C01813=1094.520,430.598,-102.360,178.831,24.503,153.665
C01814=1094.514,430.353,-102.317,178.828,24.492,153.663
C01815=1094.508,430.106,-102.276,178.825,24.481,153.660
C01816=1094.502,429.860,-102.233,178.822,24.469,153.658
C01817=1094.495,429.613,-102.192,178.819,24.459,153.656
C01818=1094.490,429.367,-102.149,178.817,24.448,153.653
C01819=1094.483,429.120,-102.107,178.813,24.437,153.651
C01820=1094.477,428.875,-102.065,178.811,24.426,153.649
C01821=1094.470,428.628,-102.023,178.808,24.416,153.646
C01822=1094.464,428.382,-101.981,178.805,24.405,153.644
C01823=1094.457,428.135,-101.939,178.802,24.394,153.642
C01824=1094.451,427.889,-101.898,178.799,24.383,153.639
C01825=1094.445,427.643,-101.855,178.797,24.373,153.637
C01826=1094.439,427.397,-101.814,178.793,24.362,153.635
C01827=1094.433,427.150,-101.772,178.791,24.352,153.633
C01828=1094.426,426.904,-101.730,178.788,24.342,153.630
C01829=1094.420,426.658,-101.688,178.785,24.331,153.628
C01830=1094.413,426.411,-101.646,178.782,24.320,153.626
C01831=1094.407,426.165,-101.605,178.779,24.310,153.624
C01832=1094.401,425.919,-101.563,178.776,24.300,153.622
C01833=1094.395,425.672,-101.522,178.774,24.289,153.619
C01834=1094.389,425.443,-101.483,178.771,24.280,153.617
C01835=1094.384,425.215,-101.444,178.768,24.270,153.615
C01836=1094.378,424.987,-101.406,178.766,24.261,153.613
C01837=1094.372,424.758,-101.367,178.763,24.251,153.611
C01838=1094.366,424.529,-101.329,178.760,24.242,153.609
C01839=1094.360,424.301,-101.290,178.757,24.232,153.607
C01840=1094.355,424.073,-101.252,178.755,24.223,153.605
C01841=1094.349,423.844,-101.213,178.752,24.214,153.603
C01842=1094.344,423.598,-101.172,178.749,24.204,153.601
C01843=1094.337,423.351,-101.130,178.746,24.194,153.599
C01844=1094.330,423.105,-101.089,178.744,24.184,153.597
C01845=1094.324,422.859,-101.047,178.741,24.174,153.595
C01846=1094.319,422.612,-101.007,178.738,24.164,153.593
C01847=1094.312,422.365,-100.965,178.734,24.154,153.591
C01848=1094.306,422.119,-100.923,178.732,24.144,153.589
C01849=1094.300,421.873,-100.883,178.729,24.134,153.587
C01850=1094.294,421.627,-100.842,178.726,24.125,153.585
C01851=1094.287,421.380,-100.800,178.723,24.115,153.583
C01852=1094.281,421.134,-100.759,178.720,24.105,153.581
C01853=1094.275,420.887,-100.718,178.717,24.095,153.579
C01854=1094.269,420.641,-100.677,178.714,24.086,153.577
C01855=1094.263,420.393,-100.636,178.712,24.076,153.575
C01856=1094.256,420.147,-100.595,178.709,24.067,153.573
C01857=1094.250,419.901,-100.553,178.706,24.057,153.571
C01858=1094.245,419.654,-100.513,178.703,24.048,153.569
C01859=1094.238,419.408,-100.472,178.700,24.038,153.567
C01860=1094.232,419.161,-100.431,178.697,24.029,153.565
C01861=1094.225,418.914,-100.391,178.694,24.019,153.563
C01862=1094.219,418.668,-100.349,178.691,24.010,153.561
C01863=1094.214,418.421,-100.308,178.689,24.000,153.559
C01864=1094.207,418.175,-100.268,178.686,23.991,153.557
C01865=1094.201,417.929,-100.227,178.683,23.982,153.555
C01866=1094.195,417.682,-100.187,178.680,23.972,153.553
C01867=1094.189,417.436,-100.145,178.677,23.963,153.551
C01868=1094.183,417.188,-100.104,178.675,23.954,153.549
C01869=1094.176,416.942,-100.064,178.672,23.945,153.548
C01870=1094.171,416.695,-100.023,178.669,23.936,153.546
C01871=1094.164,416.449,-99.982,178.666,23.926,153.544
C01872=1094.158,416.202,-99.942,178.663,23.918,153.542
C01873=1094.152,415.956,-99.901,178.660,23.908,153.540
C01874=1094.146,415.709,-99.861,178.657,23.899,153.538
C01875=1094.140,415.462,-99.821,178.654,23.890,153.536
C01876=1094.134,415.216,-99.780,178.652,23.882,153.535
C01877=1094.128,414.969,-99.740,178.649,23.873,153.533
C01878=1094.122,414.723,-99.700,178.646,23.864,153.531
C01879=1094.114,414.476,-99.658,178.643,23.855,153.529
C01880=1094.109,414.229,-99.618,178.640,23.846,153.527
C01881=1094.102,413.983,-99.577,178.636,23.837,153.526
C01882=1094.096,413.735,-99.538,178.634,23.828,153.524
C01883=1094.091,413.489,-99.497,178.631,23.820,153.522
C01884=1094.084,413.242,-99.457,178.628,23.811,153.520
C01885=1094.078,412.996,-99.417,178.625,23.802,153.519
C01886=1094.071,412.749,-99.377,178.623,23.794,153.517
C01887=1094.066,412.502,-99.336,178.620,23.785,153.515
C01888=1094.059,412.256,-99.296,178.617,23.776,153.513
C01889=1094.053,412.009,-99.256,178.614,23.768,153.512
C01890=1094.048,411.788,-99.221,178.611,23.760,153.510
C01891=1094.043,411.567,-99.184,178.609,23.753,153.509
C01892=1094.038,411.345,-99.148,178.606,23.745,153.507
C01893=1094.032,411.125,-99.112,178.604,23.737,153.506
C01894=1094.026,410.904,-99.076,178.601,23.730,153.504
C01895=1094.021,410.682,-99.041,178.599,23.722,153.503
C01896=1094.015,410.461,-99.004,178.595,23.714,153.501
C01897=1094.011,410.240,-98.969,178.593,23.706,153.499
C01898=1094.004,409.993,-98.929,178.591,23.698,153.498
C01899=1093.998,409.746,-98.889,178.588,23.690,153.496
C01900=1093.992,409.500,-98.849,178.584,23.681,153.495
C01901=1093.986,409.253,-98.808,178.582,23.673,153.493
C01902=1093.980,409.006,-98.769,178.579,23.665,153.491
C01903=1093.974,408.759,-98.729,178.576,23.656,153.490
C01904=1093.968,408.513,-98.690,178.574,23.648,153.488
C01905=1093.962,408.266,-98.650,178.570,23.640,153.486
C01906=1093.956,408.019,-98.610,178.568,23.632,153.485
C01907=1093.949,407.773,-98.570,178.565,23.624,153.483
C01908=1093.943,407.525,-98.531,178.561,23.616,153.482
C01909=1093.938,407.279,-98.491,178.559,23.607,153.480
C01910=1093.932,407.032,-98.451,178.556,23.599,153.478
C01911=1093.926,406.785,-98.411,178.554,23.591,153.477
C01912=1093.920,406.538,-98.372,178.550,23.583,153.475
C01913=1093.914,406.291,-98.332,178.547,23.575,153.474
C01914=1093.908,406.045,-98.293,178.545,23.567,153.472
C01915=1093.902,405.798,-98.253,178.542,23.559,153.470
C01916=1093.895,405.551,-98.214,178.539,23.551,153.469
C01917=1093.889,405.304,-98.174,178.536,23.543,153.467
C01918=1093.883,405.058,-98.135,178.533,23.536,153.466
C01919=1093.877,404.811,-98.096,178.530,23.528,153.464
C01920=1093.871,404.564,-98.056,178.528,23.520,153.463
C01921=1093.865,404.317,-98.017,178.524,23.512,153.461
C01922=1093.859,404.071,-97.977,178.522,23.504,153.460
C01923=1093.853,403.824,-97.938,178.519,23.497,153.458
C01924=1093.847,403.577,-97.899,178.516,23.489,153.457
C01925=1093.841,403.330,-97.860,178.513,23.481,153.455
C01926=1093.835,403.083,-97.820,178.510,23.474,153.454
C01927=1093.829,402.836,-97.781,178.507,23.466,153.452
C01928=1093.823,402.590,-97.742,178.505,23.458,153.451
C01929=1093.817,402.343,-97.703,178.501,23.450,153.449
C01930=1093.811,402.096,-97.664,178.499,23.443,153.448
C01931=1093.805,401.849,-97.625,178.496,23.435,153.446
C01932=1093.799,401.602,-97.585,178.493,23.428,153.445
C01933=1093.792,401.355,-97.546,178.490,23.421,153.444
C01934=1093.787,401.108,-97.508,178.487,23.412,153.442
C01935=1093.781,400.861,-97.468,178.485,23.405,153.441
C01936=1093.775,400.614,-97.429,178.482,23.398,153.439
C01937=1093.769,400.368,-97.391,178.479,23.390,153.438
C01938=1093.763,400.121,-97.351,178.476,23.383,153.437
C01939=1093.757,399.874,-97.312,178.473,23.376,153.435
C01940=1093.751,399.627,-97.274,178.470,23.368,153.434
C01941=1093.745,399.380,-97.235,178.468,23.361,153.432
C01942=1093.739,399.133,-97.195,178.464,23.353,153.431
C01943=1093.733,398.886,-97.157,178.462,23.346,153.430
C01944=1093.727,398.639,-97.118,178.459,23.339,153.428
C01945=1093.720,398.393,-97.079,178.456,23.332,153.427
C01946=1093.715,398.172,-97.044,178.453,23.325,153.426
C01947=1093.710,397.951,-97.010,178.451,23.319,153.424
C01948=1093.704,397.730,-96.976,178.448,23.312,153.423
C01949=1093.700,397.509,-96.941,178.446,23.306,153.422
C01950=1093.694,397.289,-96.907,178.443,23.299,153.421
C01951=1093.688,397.068,-96.872,178.441,23.293,153.420
C01952=1093.683,396.847,-96.837,178.438,23.287,153.418
C01953=1093.678,396.626,-96.803,178.435,23.280,153.417
C01954=1093.671,396.379,-96.764,178.433,23.274,153.416
C01955=1093.666,396.132,-96.726,178.430,23.266,153.415
C01956=1093.659,395.885,-96.687,178.427,23.259,153.413
C01957=1093.654,395.638,-96.649,178.424,23.252,153.412
C01958=1093.647,395.391,-96.610,178.421,23.245,153.411
C01959=1093.642,395.144,-96.572,178.418,23.238,153.409
C01960=1093.636,394.898,-96.533,178.415,23.231,153.408
C01961=1093.630,394.650,-96.494,178.413,23.224,153.407
C01962=1093.624,394.404,-96.457,178.410,23.217,153.406
C01963=1093.618,394.157,-96.418,178.406,23.210,153.404
C01964=1093.612,393.910,-96.379,178.404,23.203,153.403
C01965=1093.606,393.663,-96.342,178.401,23.197,153.402
C01966=1093.600,393.416,-96.303,178.398,23.190,153.401
C01967=1093.594,393.169,-96.265,178.395,23.183,153.399
C01968=1093.588,392.922,-96.226,178.392,23.176,153.398
C01969=1093.582,392.675,-96.189,178.389,23.169,153.397
C01970=1093.576,392.428,-96.151,178.387,23.163,153.396
C01971=1093.570,392.181,-96.111,178.384,23.156,153.394
C01972=1093.564,391.934,-96.074,178.380,23.149,153.393
C01973=1093.558,391.688,-96.036,178.378,23.142,153.392
C01974=1093.552,391.440,-95.998,178.375,23.136,153.391
C01975=1093.546,391.193,-95.960,178.372,23.130,153.390
C01976=1093.540,390.947,-95.922,178.369,23.123,153.388
C01977=1093.534,390.699,-95.884,178.366,23.116,153.387
C01978=1093.528,390.452,-95.846,178.363,23.110,153.386
C01979=1093.522,390.206,-95.807,178.360,23.103,153.385
C01980=1093.516,389.959,-95.769,178.357,23.096,153.384
C01981=1093.510,389.712,-95.732,178.355,23.090,153.383
C01982=1093.504,389.465,-95.694,178.351,23.083,153.381
C01983=1093.498,389.218,-95.656,178.348,23.076,153.380
C01984=1093.491,388.971,-95.618,178.345,23.070,153.379
C01985=1093.486,388.724,-95.581,178.343,23.064,153.378
C01986=1093.480,388.477,-95.543,178.340,23.057,153.377
C01987=1093.474,388.230,-95.505,178.337,23.051,153.376
C01988=1093.468,387.983,-95.468,178.333,23.044,153.375
C01989=1093.462,387.736,-95.429,178.331,23.038,153.373
C01990=1093.456,387.489,-95.392,178.328,23.031,153.372
C01991=1093.450,387.242,-95.354,178.325,23.025,153.371
C01992=1093.444,386.995,-95.317,178.322,23.019,153.370
C01993=1093.438,386.748,-95.279,178.319,23.013,153.369
C01994=1093.432,386.502,-95.241,178.316,23.006,153.368
C01995=1093.426,386.254,-95.203,178.314,23.000,153.367
C01996=1093.420,386.007,-95.166,178.310,22.993,153.366
C01997=1093.414,385.760,-95.128,178.307,22.987,153.365
C01998=1093.408,385.513,-95.091,178.304,22.981,153.363
C01999=1093.402,385.267,-95.053,178.301,22.975,153.362
C02000=1093.397,385.019,-95.016,178.298,22.969,153.361
C02001=1093.391,384.772,-94.978,178.296,22.962,153.360
C02002=1093.386,384.558,-94.946,178.294,22.957,153.359
C02003=1093.381,384.343,-94.913,178.290,22.951,153.358
C02004=1093.376,384.129,-94.880,178.288,22.946,153.357
C02005=1093.371,383.915,-94.848,178.285,22.940,153.356
C02006=1093.365,383.700,-94.816,178.283,22.935,153.356
C02007=1093.361,383.486,-94.783,178.281,22.930,153.355
C02008=1093.355,383.272,-94.751,178.278,22.924,153.354
C02009=1093.351,383.057,-94.719,178.276,22.919,153.353
C02010=1093.345,382.811,-94.681,178.273,22.913,153.352
C02011=1093.339,382.563,-94.644,178.270,22.907,153.351
C02012=1093.332,382.316,-94.607,178.267,22.901,153.350
C02013=1093.326,382.069,-94.569,178.264,22.895,153.349
C02014=1093.321,381.821,-94.532,178.261,22.889,153.348
C02015=1093.314,381.575,-94.495,178.258,22.883,153.347
C02016=1093.308,381.328,-94.458,178.255,22.877,153.346
C02017=1093.303,381.080,-94.421,178.252,22.871,153.345
C02018=1093.296,380.834,-94.384,178.249,22.866,153.344
C02019=1093.291,380.587,-94.347,178.245,22.859,153.343
C02020=1093.285,380.339,-94.310,178.242,22.853,153.342
C02021=1093.278,380.093,-94.273,178.239,22.847,153.341
C02022=1093.273,379.845,-94.236,178.237,22.841,153.340
C02023=1093.267,379.598,-94.199,178.234,22.836,153.339
C02024=1093.261,379.351,-94.162,178.231,22.830,153.338
C02025=1093.255,379.104,-94.125,178.228,22.824,153.337
C02026=1093.249,378.857,-94.087,178.226,22.818,153.336
C02027=1093.243,378.610,-94.051,178.222,22.813,153.335
C02028=1093.237,378.362,-94.014,178.219,22.807,153.334
C02029=1093.231,378.115,-93.977,178.217,22.801,153.333
C02030=1093.225,377.868,-93.940,178.213,22.796,153.332
C02031=1093.220,377.621,-93.903,178.210,22.790,153.331
C02032=1093.213,377.374,-93.867,178.208,22.784,153.330
C02033=1093.208,377.127,-93.830,178.204,22.778,153.329
C02034=1093.202,376.880,-93.794,178.202,22.772,153.328
C02035=1093.197,376.633,-93.757,178.198,22.767,153.327
C02036=1093.191,376.385,-93.720,178.196,22.761,153.326
C02037=1093.185,376.138,-93.683,178.192,22.755,153.325
C02038=1093.179,375.891,-93.646,178.189,22.749,153.324
C02039=1093.173,375.644,-93.610,178.186,22.744,153.323
C02040=1093.167,375.396,-93.573,178.183,22.738,153.323
C02041=1093.161,375.150,-93.537,178.180,22.732,153.322
C02042=1093.156,374.903,-93.500,178.177,22.727,153.321
C02043=1093.149,374.656,-93.463,178.175,22.722,153.320
C02044=1093.144,374.408,-93.426,178.172,22.716,153.319
C02045=1093.138,374.160,-93.390,178.169,22.710,153.318
C02046=1093.132,373.913,-93.353,178.166,22.705,153.317
C02047=1093.126,373.666,-93.317,178.163,22.699,153.316
C02048=1093.120,373.420,-93.281,178.160,22.694,153.315
C02049=1093.115,373.172,-93.244,178.157,22.688,153.315
C02050=1093.108,372.925,-93.208,178.154,22.683,153.314
C02051=1093.102,372.678,-93.172,178.150,22.677,153.313
C02052=1093.096,372.431,-93.135,178.147,22.672,153.312
C02053=1093.091,372.183,-93.099,178.145,22.667,153.311
C02054=1093.084,371.936,-93.062,178.142,22.661,153.310
C02055=1093.078,371.689,-93.026,178.139,22.656,153.309
C02056=1093.073,371.441,-92.990,178.136,22.650,153.309
C02057=1093.067,371.194,-92.953,178.133,22.645,153.308
C02058=1093.057,370.793,-92.895,178.128,22.636,153.306
C02059=1093.048,370.391,-92.836,178.123,22.627,153.305
C02060=1093.038,369.990,-92.777,178.119,22.619,153.304
C02061=1093.029,369.590,-92.719,178.114,22.610,153.302
C02062=1093.023,369.342,-92.683,178.111,22.605,153.301
C02063=1093.017,369.094,-92.647,178.107,22.600,153.301
C02064=1093.011,368.847,-92.610,178.104,22.594,153.300
C02065=1093.005,368.600,-92.575,178.101,22.589,153.299
C02066=1092.999,368.353,-92.538,178.099,22.584,153.298
C02067=1092.993,368.105,-92.503,178.096,22.579,153.297
C02068=1092.988,367.858,-92.467,178.092,22.574,153.297
C02069=1092.982,367.611,-92.430,178.089,22.568,153.296
C02070=1092.976,367.363,-92.394,178.086,22.563,153.295
C02071=1092.971,367.116,-92.359,178.084,22.558,153.294
C02072=1092.964,366.869,-92.323,178.081,22.553,153.293
C02073=1092.958,366.622,-92.287,178.077,22.548,153.293
C02074=1092.954,366.374,-92.251,178.074,22.542,153.292
C02075=1092.948,366.127,-92.215,178.071,22.537,153.291
C02076=1092.941,365.880,-92.179,178.069,22.532,153.290
C02077=1092.936,365.633,-92.143,178.066,22.527,153.289
C02078=1092.930,365.385,-92.108,178.062,22.522,153.289
C02079=1092.924,365.137,-92.072,178.059,22.517,153.288
C02080=1092.918,364.890,-92.037,178.056,22.512,153.287
C02081=1092.912,364.643,-92.000,178.054,22.507,153.287
C02082=1092.906,364.396,-91.964,178.050,22.502,153.286
C02083=1092.900,364.149,-91.929,178.047,22.497,153.285
C02084=1092.894,363.901,-91.893,178.044,22.491,153.284
C02085=1092.889,363.654,-91.858,178.042,22.487,153.284
C02086=1092.883,363.406,-91.822,178.038,22.482,153.283
C02087=1092.876,363.159,-91.787,178.035,22.477,153.282
C02088=1092.871,362.912,-91.752,178.032,22.471,153.281
C02089=1092.865,362.664,-91.716,178.029,22.467,153.281
C02090=1092.859,362.417,-91.681,178.026,22.462,153.280
C02091=1092.853,362.170,-91.645,178.023,22.457,153.279
C02092=1092.847,361.922,-91.609,178.020,22.452,153.279
C02093=1092.842,361.675,-91.574,178.017,22.447,153.278
C02094=1092.836,361.427,-91.538,178.014,22.442,153.277
C02095=1092.831,361.180,-91.503,178.011,22.437,153.276
C02096=1092.824,360.932,-91.468,178.008,22.433,153.276
C02097=1092.818,360.685,-91.433,178.005,22.428,153.275
C02098=1092.812,360.438,-91.397,178.002,22.423,153.274
C02099=1092.807,360.191,-91.362,177.999,22.418,153.274
C02100=1092.801,359.943,-91.326,177.996,22.414,153.273
C02101=1092.795,359.695,-91.292,177.993,22.408,153.272
C02102=1092.789,359.448,-91.256,177.990,22.403,153.271
C02103=1092.783,359.200,-91.221,177.987,22.399,153.271
C02104=1092.778,358.953,-91.185,177.984,22.394,153.270
C02105=1092.771,358.705,-91.151,177.980,22.389,153.270
C02106=1092.766,358.458,-91.115,177.978,22.385,153.269
C02107=1092.760,358.211,-91.080,177.975,22.380,153.268
C02108=1092.754,357.963,-91.046,177.971,22.375,153.267
C02109=1092.748,357.716,-91.010,177.969,22.371,153.267
C02110=1092.739,357.330,-90.955,177.963,22.363,153.266
C02111=1092.730,356.944,-90.901,177.959,22.356,153.265
C02112=1092.721,356.558,-90.846,177.955,22.349,153.264
C02113=1092.712,356.172,-90.791,177.950,22.342,153.263
C02114=1092.706,355.925,-90.757,177.947,22.337,153.262
C02115=1092.700,355.678,-90.722,177.943,22.332,153.261
C02116=1092.695,355.429,-90.687,177.941,22.328,153.261
C02117=1092.688,355.183,-90.652,177.937,22.323,153.260
C02118=1092.683,354.935,-90.617,177.934,22.318,153.260
C02119=1092.677,354.688,-90.582,177.932,22.314,153.259
C02120=1092.671,354.440,-90.547,177.928,22.309,153.258
C02121=1092.666,354.192,-90.512,177.925,22.304,153.258
C02122=1092.659,353.945,-90.478,177.922,22.300,153.257
C02123=1092.654,353.697,-90.443,177.919,22.295,153.256
C02124=1092.648,353.449,-90.408,177.916,22.291,153.256
C02125=1092.642,353.203,-90.373,177.913,22.286,153.255
C02126=1092.637,352.955,-90.339,177.910,22.282,153.255
C02127=1092.631,352.707,-90.304,177.907,22.277,153.254
C02128=1092.625,352.460,-90.269,177.904,22.273,153.253
C02129=1092.619,352.212,-90.234,177.901,22.269,153.253
C02130=1092.613,351.965,-90.200,177.898,22.264,153.252
C02131=1092.608,351.717,-90.166,177.894,22.259,153.252
C02132=1092.601,351.470,-90.130,177.892,22.255,153.251
C02133=1092.595,351.222,-90.096,177.889,22.250,153.250
C02134=1092.586,350.816,-90.040,177.884,22.243,153.249
C02135=1092.576,350.409,-89.983,177.879,22.236,153.249
C02136=1092.566,350.002,-89.926,177.874,22.229,153.248
C02137=1092.557,349.596,-89.870,177.869,22.221,153.247
C02138=1092.552,349.348,-89.835,177.865,22.217,153.246
C02139=1092.546,349.101,-89.801,177.863,22.213,153.245
C02140=1092.540,348.853,-89.767,177.859,22.208,153.245
C02141=1092.534,348.605,-89.732,177.856,22.204,153.244
C02142=1092.529,348.358,-89.698,177.853,22.199,153.244
C02143=1092.523,348.111,-89.664,177.851,22.195,153.243
C02144=1092.518,347.863,-89.629,177.847,22.191,153.243
C02145=1092.511,347.615,-89.595,177.844,22.187,153.242
C02146=1092.505,347.368,-89.561,177.841,22.182,153.242
C02147=1092.500,347.120,-89.526,177.838,22.178,153.241
C02148=1092.494,346.873,-89.492,177.835,22.174,153.241
C02149=1092.488,346.625,-89.458,177.832,22.169,153.240
C02150=1092.482,346.377,-89.424,177.829,22.165,153.239
C02151=1092.477,346.129,-89.390,177.825,22.161,153.239
C02152=1092.471,345.882,-89.356,177.823,22.157,153.238
C02153=1092.465,345.635,-89.322,177.819,22.152,153.238
C02154=1092.459,345.387,-89.287,177.817,22.148,153.237
C02155=1092.453,345.139,-89.254,177.813,22.144,153.237
C02156=1092.448,344.891,-89.219,177.811,22.140,153.236
C02157=1092.442,344.644,-89.185,177.807,22.135,153.236
C02158=1092.436,344.408,-89.153,177.805,22.132,153.235
C02159=1092.431,344.172,-89.120,177.802,22.128,153.235
C02160=1092.426,343.935,-89.088,177.798,22.124,153.234
C02161=1092.420,343.700,-89.056,177.796,22.119,153.234
C02162=1092.414,343.464,-89.023,177.793,22.116,153.233
C02163=1092.408,343.229,-88.991,177.790,22.112,153.233
C02164=1092.403,342.992,-88.959,177.787,22.108,153.232
C02165=1092.398,342.756,-88.927,177.784,22.104,153.232
C02166=1092.392,342.509,-88.893,177.781,22.100,153.231
C02167=1092.386,342.260,-88.859,177.778,22.096,153.231
C02168=1092.380,342.013,-88.825,177.775,22.092,153.230
C02169=1092.375,341.765,-88.792,177.772,22.088,153.230
C02170=1092.369,341.518,-88.758,177.769,22.084,153.229
C02171=1092.363,341.270,-88.724,177.766,22.079,153.229
C02172=1092.357,341.023,-88.690,177.763,22.075,153.228
C02173=1092.352,340.775,-88.657,177.759,22.071,153.228
C02174=1092.346,340.527,-88.623,177.757,22.067,153.227
C02175=1092.340,340.280,-88.589,177.753,22.063,153.227
C02176=1092.334,340.032,-88.555,177.751,22.059,153.226
C02177=1092.328,339.784,-88.522,177.747,22.055,153.226
C02178=1092.322,339.536,-88.488,177.744,22.051,153.225
C02179=1092.317,339.288,-88.454,177.742,22.047,153.225
C02180=1092.311,339.041,-88.421,177.738,22.043,153.225
C02181=1092.305,338.793,-88.387,177.735,22.039,153.224
C02182=1092.300,338.545,-88.354,177.732,22.035,153.224
C02183=1092.294,338.298,-88.321,177.729,22.031,153.223
C02184=1092.288,338.051,-88.287,177.726,22.027,153.223
C02185=1092.282,337.803,-88.253,177.723,22.023,153.222
C02186=1092.277,337.555,-88.220,177.720,22.019,153.222
C02187=1092.271,337.307,-88.187,177.717,22.015,153.221
C02188=1092.265,337.060,-88.153,177.714,22.011,153.221
C02189=1092.259,336.812,-88.120,177.710,22.007,153.220
C02190=1092.253,336.564,-88.087,177.708,22.003,153.220
C02191=1092.248,336.316,-88.053,177.704,21.999,153.220
C02192=1092.242,336.068,-88.020,177.701,21.995,153.219
C02193=1092.236,335.821,-87.986,177.698,21.992,153.219
C02194=1092.230,335.573,-87.953,177.695,21.988,153.218
C02195=1092.225,335.325,-87.920,177.692,21.984,153.218
C02196=1092.219,335.078,-87.886,177.689,21.980,153.217
C02197=1092.213,334.830,-87.854,177.686,21.976,153.217
C02198=1092.207,334.582,-87.820,177.683,21.972,153.216
C02199=1092.202,334.334,-87.787,177.680,21.969,153.216
C02200=1092.195,334.087,-87.754,177.677,21.965,153.216
C02201=1092.190,333.839,-87.721,177.674,21.961,153.215
C02202=1092.184,333.591,-87.688,177.671,21.957,153.215
C02203=1092.179,333.343,-87.654,177.668,21.954,153.214
C02204=1092.172,333.095,-87.622,177.664,21.949,153.214
C02205=1092.167,332.848,-87.589,177.661,21.946,153.214
C02206=1092.162,332.600,-87.555,177.659,21.942,153.213
C02207=1092.156,332.353,-87.522,177.655,21.938,153.213
C02208=1092.150,332.105,-87.489,177.652,21.934,153.212
C02209=1092.144,331.857,-87.456,177.650,21.930,153.212
C02210=1092.138,331.609,-87.423,177.646,21.927,153.212
C02211=1092.132,331.362,-87.390,177.643,21.923,153.211
C02212=1092.126,331.114,-87.357,177.640,21.920,153.211
C02213=1092.120,330.866,-87.324,177.637,21.915,153.210
C02214=1092.111,330.477,-87.273,177.632,21.910,153.210
C02215=1092.102,330.087,-87.222,177.628,21.905,153.209
C02216=1092.093,329.698,-87.170,177.623,21.898,153.209
C02217=1092.083,329.308,-87.119,177.618,21.893,153.208
C02218=1092.078,329.061,-87.085,177.615,21.889,153.208
C02219=1092.072,328.813,-87.053,177.611,21.885,153.207
C02220=1092.066,328.565,-87.021,177.608,21.882,153.207
C02221=1092.061,328.318,-86.988,177.605,21.879,153.207
C02222=1092.054,328.070,-86.955,177.602,21.874,153.206
C02223=1092.049,327.821,-86.922,177.599,21.871,153.206
C02224=1092.043,327.574,-86.889,177.596,21.868,153.205
C02225=1092.036,327.326,-86.857,177.593,21.864,153.205
C02226=1092.031,327.078,-86.824,177.590,21.860,153.205
C02227=1092.026,326.831,-86.792,177.587,21.857,153.204
C02228=1092.020,326.583,-86.760,177.584,21.853,153.204
C02229=1092.014,326.335,-86.726,177.580,21.849,153.204
C02230=1092.008,326.086,-86.694,177.577,21.846,153.203
C02231=1092.002,325.839,-86.662,177.575,21.842,153.203
C02232=1091.996,325.592,-86.629,177.571,21.838,153.203
C02233=1091.991,325.343,-86.597,177.568,21.835,153.202
C02234=1091.984,325.096,-86.564,177.565,21.832,153.202
C02235=1091.978,324.848,-86.532,177.563,21.828,153.201
C02236=1091.974,324.600,-86.500,177.559,21.824,153.201
C02237=1091.968,324.352,-86.467,177.556,21.821,153.201
C02238=1091.962,324.104,-86.435,177.553,21.817,153.200
C02239=1091.956,323.857,-86.402,177.550,21.814,153.200
C02240=1091.951,323.609,-86.370,177.547,21.810,153.200
C02241=1091.945,323.360,-86.338,177.544,21.807,153.199
C02242=1091.938,323.113,-86.305,177.541,21.803,153.199
C02243=1091.933,322.865,-86.273,177.538,21.800,153.199
C02244=1091.927,322.617,-86.240,177.534,21.796,153.198
C02245=1091.921,322.369,-86.208,177.532,21.792,153.198
C02246=1091.916,322.122,-86.176,177.529,21.789,153.198
C02247=1091.910,321.873,-86.144,177.526,21.786,153.197
C02248=1091.904,321.626,-86.111,177.522,21.782,153.197
C02249=1091.899,321.378,-86.079,177.519,21.779,153.197
C02250=1091.893,321.130,-86.047,177.517,21.775,153.196
C02251=1091.888,320.882,-86.016,177.514,21.772,153.196
C02252=1091.881,320.635,-85.983,177.510,21.768,153.196
C02253=1091.876,320.386,-85.950,177.507,21.764,153.195
C02254=1091.871,320.139,-85.919,177.504,21.761,153.195
C02255=1091.865,319.890,-85.887,177.502,21.758,153.195
C02256=1091.859,319.643,-85.855,177.498,21.754,153.194
C02257=1091.853,319.395,-85.823,177.495,21.751,153.194
C02258=1091.848,319.148,-85.790,177.492,21.747,153.194
C02259=1091.842,318.900,-85.758,177.489,21.744,153.193
C02260=1091.837,318.651,-85.726,177.486,21.741,153.193
C02261=1091.831,318.404,-85.694,177.483,21.737,153.193
C02262=1091.825,318.155,-85.662,177.480,21.733,153.192
C02263=1091.820,317.908,-85.630,177.477,21.730,153.192
C02264=1091.814,317.660,-85.598,177.474,21.727,153.192
C02265=1091.808,317.412,-85.567,177.470,21.723,153.191
C02266=1091.799,317.016,-85.515,177.466,21.718,153.191
C02267=1091.791,316.620,-85.465,177.461,21.712,153.190
C02268=1091.782,316.224,-85.413,177.456,21.706,153.190
C02269=1091.773,315.827,-85.363,177.452,21.702,153.189
C02270=1091.767,315.579,-85.331,177.448,21.698,153.189
C02271=1091.761,315.332,-85.300,177.445,21.694,153.189
C02272=1091.755,315.083,-85.268,177.442,21.691,153.189
C02273=1091.750,314.836,-85.236,177.439,21.688,153.188
C02274=1091.744,314.587,-85.205,177.436,21.685,153.188
C02275=1091.739,314.339,-85.173,177.433,21.682,153.188
C02276=1091.732,314.092,-85.142,177.430,21.678,153.187
C02277=1091.727,313.844,-85.110,177.427,21.675,153.187
C02278=1091.721,313.596,-85.078,177.424,21.672,153.187
C02279=1091.715,313.347,-85.047,177.421,21.668,153.187
C02280=1091.709,313.100,-85.016,177.418,21.665,153.186
C02281=1091.703,312.852,-84.984,177.415,21.662,153.186
C02282=1091.698,312.604,-84.952,177.411,21.659,153.186
C02283=1091.691,312.356,-84.921,177.408,21.655,153.186
C02284=1091.686,312.108,-84.890,177.405,21.652,153.185
C02285=1091.680,311.861,-84.858,177.402,21.649,153.185
C02286=1091.674,311.612,-84.827,177.399,21.646,153.185
C02287=1091.669,311.364,-84.795,177.396,21.643,153.185
C02288=1091.663,311.116,-84.763,177.393,21.639,153.184
C02289=1091.657,310.868,-84.733,177.390,21.636,153.184
C02290=1091.651,310.620,-84.701,177.387,21.633,153.184
C02291=1091.645,310.373,-84.669,177.384,21.630,153.183
C02292=1091.640,310.125,-84.639,177.381,21.627,153.183
C02293=1091.634,309.877,-84.607,177.378,21.623,153.183
C02294=1091.628,309.629,-84.577,177.375,21.621,153.183
C02295=1091.622,309.381,-84.545,177.371,21.617,153.183
C02296=1091.617,309.133,-84.514,177.368,21.614,153.182
C02297=1091.611,308.885,-84.483,177.365,21.611,153.182
C02298=1091.605,308.636,-84.451,177.362,21.608,153.182
C02299=1091.599,308.389,-84.420,177.359,21.604,153.182
C02300=1091.594,308.141,-84.389,177.356,21.602,153.181
C02301=1091.588,307.893,-84.357,177.353,21.598,153.181
C02302=1091.582,307.645,-84.327,177.350,21.595,153.181
C02303=1091.577,307.398,-84.295,177.347,21.591,153.181
C02304=1091.570,307.149,-84.265,177.344,21.589,153.180
C02305=1091.565,306.902,-84.233,177.341,21.585,153.180
C02306=1091.559,306.654,-84.203,177.338,21.582,153.180
C02307=1091.553,306.405,-84.171,177.335,21.579,153.180
C02308=1091.547,306.158,-84.140,177.332,21.576,153.179
C02309=1091.542,305.910,-84.109,177.329,21.573,153.179
C02310=1091.537,305.661,-84.078,177.326,21.570,153.179
C02311=1091.530,305.414,-84.047,177.322,21.567,153.179
C02312=1091.525,305.165,-84.016,177.319,21.563,153.178
C02313=1091.519,304.918,-83.986,177.316,21.560,153.178
C02314=1091.514,304.669,-83.955,177.313,21.557,153.178
C02315=1091.508,304.422,-83.923,177.310,21.554,153.178
C02316=1091.502,304.173,-83.892,177.307,21.551,153.177
C02317=1091.497,303.926,-83.862,177.304,21.548,153.177
C02318=1091.488,303.532,-83.813,177.299,21.543,153.177
C02319=1091.479,303.138,-83.763,177.295,21.538,153.176
C02320=1091.470,302.746,-83.715,177.289,21.533,153.176
C02321=1091.461,302.352,-83.667,177.285,21.528,153.176
C02322=1091.455,302.103,-83.636,177.282,21.525,153.175
C02323=1091.449,301.856,-83.604,177.279,21.522,153.175
C02324=1091.444,301.608,-83.574,177.275,21.519,153.175
C02325=1091.439,301.360,-83.543,177.272,21.515,153.175
C02326=1091.433,301.112,-83.513,177.269,21.513,153.175
C02327=1091.427,300.864,-83.482,177.266,21.509,153.174
C02328=1091.422,300.616,-83.451,177.263,21.506,153.174
C02329=1091.416,300.368,-83.421,177.260,21.503,153.174
C02330=1091.410,300.119,-83.390,177.257,21.500,153.174
C02331=1091.405,299.871,-83.359,177.254,21.497,153.173
C02332=1091.399,299.624,-83.329,177.251,21.494,153.173
C02333=1091.394,299.376,-83.298,177.248,21.491,153.173
C02334=1091.388,299.128,-83.268,177.245,21.488,153.173
C02335=1091.383,298.880,-83.237,177.242,21.485,153.173
C02336=1091.377,298.631,-83.207,177.239,21.482,153.172
C02337=1091.371,298.383,-83.177,177.236,21.479,153.172
C02338=1091.366,298.135,-83.146,177.233,21.476,153.172
C02339=1091.361,297.887,-83.115,177.231,21.473,153.172
C02340=1091.355,297.640,-83.085,177.227,21.469,153.171
C02341=1091.349,297.392,-83.055,177.224,21.467,153.171
C02342=1091.342,297.143,-83.024,177.221,21.464,153.171
C02343=1091.337,296.895,-82.994,177.218,21.461,153.171
C02344=1091.332,296.647,-82.963,177.214,21.458,153.171
C02345=1091.326,296.399,-82.933,177.211,21.455,153.171
C02346=1091.320,296.151,-82.903,177.209,21.452,153.170
C02347=1091.315,295.903,-82.873,177.206,21.449,153.170
C02348=1091.309,295.655,-82.843,177.202,21.446,153.170
C02349=1091.303,295.407,-82.812,177.199,21.443,153.170
C02350=1091.297,295.159,-82.782,177.196,21.440,153.170
C02351=1091.292,294.911,-82.752,177.193,21.437,153.169
C02352=1091.286,294.663,-82.722,177.190,21.434,153.169
C02353=1091.280,294.415,-82.692,177.187,21.431,153.169
C02354=1091.275,294.167,-82.662,177.184,21.429,153.169
C02355=1091.269,293.919,-82.632,177.181,21.426,153.169
C02356=1091.263,293.670,-82.602,177.178,21.423,153.169
C02357=1091.257,293.422,-82.572,177.175,21.420,153.168
C02358=1091.252,293.174,-82.541,177.172,21.417,153.168
C02359=1091.247,292.926,-82.511,177.169,21.414,153.168
C02360=1091.241,292.678,-82.481,177.166,21.411,153.168
C02361=1091.236,292.430,-82.451,177.163,21.408,153.168
C02362=1091.230,292.182,-82.421,177.160,21.406,153.167
C02363=1091.224,291.934,-82.392,177.157,21.403,153.167
C02364=1091.218,291.686,-82.361,177.154,21.400,153.167
C02365=1091.212,291.437,-82.332,177.151,21.397,153.167
C02366=1091.206,291.190,-82.301,177.148,21.394,153.167
C02367=1091.201,290.941,-82.272,177.145,21.391,153.167
C02368=1091.195,290.693,-82.241,177.142,21.388,153.166
C02369=1091.190,290.445,-82.212,177.139,21.385,153.166
C02370=1091.181,290.065,-82.166,177.134,21.381,153.166
C02371=1091.172,289.686,-82.121,177.129,21.377,153.166
C02372=1091.164,289.306,-82.075,177.125,21.372,153.165
C02373=1091.155,288.927,-82.029,177.120,21.368,153.165
C02374=1091.149,288.679,-82.000,177.117,21.365,153.165
C02375=1091.144,288.430,-81.970,177.114,21.362,153.165
C02376=1091.137,288.182,-81.941,177.111,21.359,153.165
C02377=1091.132,287.934,-81.911,177.108,21.356,153.165
C02378=1091.126,287.686,-81.881,177.105,21.354,153.165
C02379=1091.121,287.437,-81.851,177.102,21.351,153.164
C02380=1091.114,287.189,-81.822,177.099,21.348,153.164
C02381=1091.108,286.942,-81.792,177.096,21.345,153.164
C02382=1091.103,286.693,-81.762,177.093,21.342,153.164
C02383=1091.098,286.445,-81.733,177.090,21.340,153.164
C02384=1091.092,286.197,-81.704,177.087,21.337,153.163
C02385=1091.086,285.949,-81.674,177.083,21.334,153.163
C02386=1091.080,285.701,-81.644,177.080,21.331,153.163
C02387=1091.075,285.453,-81.614,177.077,21.328,153.163
C02388=1091.069,285.204,-81.585,177.074,21.326,153.163
C02389=1091.063,284.956,-81.556,177.071,21.323,153.163
C02390=1091.058,284.708,-81.526,177.069,21.320,153.163
C02391=1091.052,284.460,-81.497,177.066,21.318,153.163
C02392=1091.047,284.212,-81.468,177.063,21.315,153.162
C02393=1091.041,283.963,-81.438,177.060,21.312,153.162
C02394=1091.035,283.715,-81.409,177.057,21.309,153.162
C02395=1091.030,283.467,-81.380,177.054,21.306,153.162
C02396=1091.024,283.219,-81.350,177.051,21.303,153.162
C02397=1091.018,282.971,-81.321,177.048,21.301,153.162
C02398=1091.013,282.722,-81.291,177.044,21.298,153.161
C02399=1091.007,282.474,-81.262,177.041,21.295,153.161
C02400=1091.001,282.226,-81.233,177.038,21.292,153.161
C02401=1090.996,281.978,-81.204,177.035,21.289,153.161
C02402=1090.990,281.730,-81.174,177.032,21.287,153.161
C02403=1090.984,281.481,-81.145,177.029,21.284,153.161
C02404=1090.979,281.234,-81.116,177.027,21.282,153.161
C02405=1090.973,280.986,-81.087,177.024,21.279,153.160
C02406=1090.968,280.736,-81.058,177.021,21.276,153.160
C02407=1090.962,280.488,-81.029,177.018,21.273,153.160
C02408=1090.957,280.241,-80.999,177.015,21.271,153.160
C02409=1090.950,279.992,-80.970,177.011,21.268,153.160
C02410=1090.945,279.744,-80.941,177.008,21.265,153.160
C02411=1090.939,279.495,-80.912,177.005,21.262,153.160
C02412=1090.934,279.248,-80.883,177.002,21.259,153.159
C02413=1090.928,278.999,-80.854,176.999,21.257,153.159
C02414=1090.922,278.751,-80.824,176.997,21.255,153.159
C02415=1090.917,278.503,-80.796,176.994,21.252,153.159
C02416=1090.911,278.255,-80.767,176.991,21.249,153.159
C02417=1090.905,278.006,-80.738,176.988,21.246,153.159
C02418=1090.899,277.758,-80.709,176.985,21.244,153.159
C02419=1090.894,277.510,-80.680,176.981,21.241,153.159
C02420=1090.888,277.262,-80.651,176.978,21.238,153.159
C02421=1090.883,277.013,-80.621,176.975,21.235,153.158
C02422=1090.874,276.643,-80.579,176.970,21.231,153.158
C02423=1090.866,276.273,-80.536,176.967,21.228,153.158
C02424=1090.857,275.903,-80.493,176.962,21.224,153.158
C02425=1090.848,275.533,-80.450,176.957,21.220,153.158
C02426=1090.843,275.285,-80.421,176.954,21.217,153.158
C02427=1090.838,275.036,-80.393,176.951,21.214,153.157
C02428=1090.831,274.788,-80.364,176.949,21.212,153.157
C02429=1090.827,274.540,-80.335,176.946,21.209,153.157
C02430=1090.820,274.292,-80.306,176.943,21.206,153.157
C02431=1090.815,274.044,-80.278,176.940,21.204,153.157
C02432=1090.809,273.795,-80.249,176.937,21.201,153.157
C02433=1090.804,273.546,-80.220,176.933,21.199,153.157
C02434=1090.798,273.298,-80.192,176.930,21.196,153.157
C02435=1090.792,273.050,-80.163,176.928,21.194,153.157
C02436=1090.787,272.802,-80.135,176.925,21.191,153.156
C02437=1090.781,272.554,-80.106,176.922,21.188,153.156
C02438=1090.775,272.305,-80.077,176.919,21.185,153.156
C02439=1090.770,272.057,-80.049,176.916,21.183,153.156
C02440=1090.764,271.809,-80.020,176.912,21.180,153.156
C02441=1090.758,271.561,-79.992,176.909,21.177,153.156
C02442=1090.752,271.312,-79.964,176.907,21.175,153.156
C02443=1090.747,271.064,-79.934,176.904,21.172,153.156
C02444=1090.741,270.816,-79.906,176.901,21.170,153.156
C02445=1090.736,270.567,-79.878,176.898,21.167,153.155
C02446=1090.730,270.319,-79.849,176.894,21.165,153.155
C02447=1090.724,270.071,-79.821,176.891,21.162,153.155
C02448=1090.719,269.823,-79.793,176.889,21.160,153.155
C02449=1090.713,269.574,-79.765,176.886,21.157,153.155
C02450=1090.708,269.325,-79.736,176.883,21.154,153.155
C02451=1090.702,269.077,-79.707,176.880,21.152,153.155
C02452=1090.696,268.829,-79.679,176.876,21.149,153.155
C02453=1090.691,268.580,-79.651,176.873,21.146,153.155
C02454=1090.685,268.332,-79.623,176.871,21.144,153.155
C02455=1090.679,268.084,-79.595,176.868,21.141,153.154
C02456=1090.673,267.835,-79.566,176.865,21.139,153.154
C02457=1090.668,267.587,-79.538,176.862,21.136,153.154
C02458=1090.662,267.339,-79.509,176.859,21.134,153.154
C02459=1090.656,267.091,-79.481,176.856,21.131,153.154
C02460=1090.651,266.843,-79.453,176.853,21.129,153.154
C02461=1090.645,266.594,-79.425,176.850,21.126,153.154
C02462=1090.640,266.346,-79.397,176.847,21.123,153.154
C02463=1090.634,266.097,-79.369,176.844,21.121,153.154
C02464=1090.628,265.849,-79.341,176.841,21.118,153.154
C02465=1090.623,265.600,-79.312,176.838,21.116,153.153
C02466=1090.617,265.352,-79.284,176.835,21.113,153.153
C02467=1090.611,265.103,-79.256,176.832,21.111,153.153
C02468=1090.606,264.855,-79.228,176.829,21.108,153.153
C02469=1090.601,264.607,-79.200,176.826,21.105,153.153
C02470=1090.595,264.359,-79.172,176.824,21.103,153.153
C02471=1090.589,264.111,-79.145,176.820,21.101,153.153
C02472=1090.583,263.862,-79.116,176.817,21.098,153.153
C02473=1090.577,263.614,-79.088,176.814,21.095,153.153
C02474=1090.569,263.246,-79.047,176.810,21.092,153.153
C02475=1090.560,262.879,-79.006,176.805,21.088,153.153
C02476=1090.551,262.512,-78.966,176.801,21.084,153.152
C02477=1090.543,262.145,-78.924,176.797,21.081,153.152
C02478=1090.537,261.896,-78.896,176.794,21.078,153.152
C02479=1090.531,261.648,-78.868,176.790,21.076,153.152
C02480=1090.526,261.399,-78.841,176.787,21.073,153.152
C02481=1090.520,261.151,-78.813,176.785,21.071,153.152
C02482=1090.514,260.903,-78.785,176.782,21.069,153.152
C02483=1090.508,260.654,-78.757,176.779,21.066,153.152
C02484=1090.502,260.405,-78.730,176.776,21.063,153.152
C02485=1090.497,260.157,-78.702,176.773,21.061,153.152
C02486=1090.491,259.909,-78.674,176.770,21.059,153.152
C02487=1090.485,259.660,-78.647,176.767,21.056,153.152
C02488=1090.479,259.412,-78.619,176.764,21.054,153.152
C02489=1090.474,259.163,-78.591,176.761,21.052,153.152
C02490=1090.468,258.915,-78.564,176.758,21.049,153.152
C02491=1090.462,258.666,-78.536,176.755,21.046,153.151
C02492=1090.457,258.418,-78.508,176.752,21.044,153.151
C02493=1090.451,258.170,-78.481,176.749,21.041,153.151
C02494=1090.445,257.921,-78.453,176.746,21.039,153.151
C02495=1090.440,257.673,-78.426,176.743,21.037,153.151
C02496=1090.434,257.425,-78.398,176.740,21.034,153.151
C02497=1090.429,257.175,-78.371,176.737,21.032,153.151
C02498=1090.422,256.928,-78.343,176.735,21.029,153.151
C02499=1090.417,256.679,-78.316,176.731,21.027,153.151
C02500=1090.411,256.431,-78.289,176.728,21.024,153.151
C02501=1090.406,256.182,-78.261,176.725,21.021,153.151
C02502=1090.400,255.934,-78.233,176.723,21.019,153.151
C02503=1090.395,255.685,-78.206,176.720,21.017,153.151
C02504=1090.389,255.437,-78.178,176.716,21.014,153.150
C02505=1090.383,255.188,-78.151,176.713,21.012,153.150
C02506=1090.378,254.940,-78.123,176.711,21.010,153.150
C02507=1090.372,254.692,-78.097,176.708,21.007,153.150
C02508=1090.367,254.443,-78.070,176.705,21.004,153.150
C02509=1090.360,254.195,-78.042,176.702,21.002,153.150
C02510=1090.355,253.946,-78.015,176.699,21.000,153.150
C02511=1090.350,253.698,-77.987,176.696,20.997,153.150
C02512=1090.344,253.450,-77.960,176.693,20.995,153.150
C02513=1090.338,253.200,-77.932,176.690,20.993,153.150
C02514=1090.333,252.952,-77.906,176.687,20.990,153.150
C02515=1090.327,252.704,-77.878,176.684,20.987,153.150
C02516=1090.321,252.456,-77.851,176.681,20.985,153.150
C02517=1090.316,252.207,-77.824,176.679,20.983,153.150
C02518=1090.310,251.959,-77.796,176.676,20.980,153.150
C02519=1090.305,251.710,-77.769,176.672,20.978,153.150
C02520=1090.299,251.461,-77.742,176.670,20.975,153.149
C02521=1090.294,251.213,-77.715,176.667,20.973,153.149
C02522=1090.288,250.964,-77.688,176.664,20.970,153.149
C02523=1090.283,250.716,-77.660,176.661,20.967,153.149
C02524=1090.277,250.468,-77.634,176.658,20.965,153.149
C02525=1090.271,250.220,-77.607,176.655,20.963,153.149
C02526=1090.263,249.849,-77.566,176.650,20.959,153.149
C02527=1090.255,249.479,-77.526,176.647,20.956,153.149
C02528=1090.247,249.108,-77.486,176.642,20.952,153.149
C02529=1090.238,248.739,-77.446,176.638,20.948,153.149
C02530=1090.233,248.490,-77.419,176.635,20.945,153.148
C02531=1090.227,248.242,-77.392,176.633,20.944,153.148
C02532=1090.222,247.993,-77.365,176.629,20.941,153.148
C02533=1090.217,247.745,-77.338,176.626,20.938,153.148
C02534=1090.211,247.496,-77.311,176.623,20.936,153.148
C02535=1090.205,247.247,-77.284,176.621,20.934,153.148
C02536=1090.199,246.998,-77.257,176.618,20.931,153.148
C02537=1090.194,246.750,-77.231,176.615,20.928,153.148
C02538=1090.189,246.501,-77.203,176.612,20.926,153.148
C02539=1090.183,246.253,-77.177,176.609,20.924,153.148
C02540=1090.177,246.005,-77.150,176.606,20.922,153.148
C02541=1090.171,245.756,-77.124,176.604,20.919,153.148
C02542=1090.166,245.508,-77.096,176.600,20.917,153.148
C02543=1090.160,245.259,-77.070,176.597,20.914,153.148
C02544=1090.155,245.011,-77.043,176.595,20.912,153.148
C02545=1090.149,244.763,-77.016,176.592,20.909,153.148
C02546=1090.144,244.513,-76.990,176.589,20.907,153.147
C02547=1090.138,244.265,-76.963,176.586,20.905,153.147
C02548=1090.133,244.017,-76.937,176.583,20.903,153.147
C02549=1090.127,243.768,-76.910,176.580,20.900,153.147
C02550=1090.121,243.520,-76.883,176.578,20.898,153.147
C02551=1090.115,243.271,-76.857,176.574,20.895,153.147
C02552=1090.111,243.022,-76.830,176.571,20.893,153.147
C02553=1090.105,242.774,-76.803,176.569,20.891,153.147
C02554=1090.099,242.525,-76.777,176.566,20.888,153.147
C02555=1090.093,242.277,-76.750,176.563,20.886,153.147
C02556=1090.088,242.028,-76.724,176.560,20.884,153.147
C02557=1090.082,241.780,-76.698,176.557,20.881,153.147
C02558=1090.076,241.531,-76.671,176.554,20.879,153.147
C02559=1090.071,241.282,-76.645,176.551,20.877,153.147
C02560=1090.065,241.034,-76.618,176.548,20.874,153.147
C02561=1090.059,240.786,-76.592,176.545,20.871,153.147
C02562=1090.054,240.537,-76.566,176.543,20.869,153.147
C02563=1090.048,240.288,-76.539,176.540,20.867,153.147
C02564=1090.042,240.040,-76.512,176.537,20.865,153.147
C02565=1090.037,239.791,-76.487,176.534,20.863,153.147
C02566=1090.031,239.543,-76.460,176.531,20.860,153.147
C02567=1090.025,239.294,-76.434,176.528,20.858,153.147
C02568=1090.020,239.045,-76.407,176.525,20.855,153.146
C02569=1090.014,238.797,-76.381,176.522,20.853,153.146
C02570=1090.008,238.548,-76.355,176.520,20.851,153.146
C02571=1090.003,238.300,-76.328,176.517,20.848,153.146
C02572=1089.996,238.051,-76.303,176.513,20.846,153.146
C02573=1089.991,237.803,-76.276,176.511,20.844,153.146
C02574=1089.985,237.554,-76.250,176.508,20.842,153.146
C02575=1089.980,237.306,-76.224,176.506,20.839,153.146
C02576=1089.975,237.057,-76.198,176.502,20.837,153.146
C02577=1089.969,236.809,-76.171,176.499,20.834,153.146
C02578=1089.960,236.431,-76.132,176.495,20.831,153.146
C02579=1089.952,236.054,-76.092,176.490,20.827,153.146
C02580=1089.944,235.677,-76.053,176.486,20.824,153.146
C02581=1089.935,235.300,-76.013,176.482,20.820,153.146
C02582=1089.929,235.051,-75.987,176.479,20.818,153.146
C02583=1089.924,234.802,-75.961,176.476,20.816,153.146
C02584=1089.918,234.554,-75.935,176.474,20.814,153.146
C02585=1089.912,234.305,-75.909,176.471,20.811,153.145
C02586=1089.908,234.057,-75.883,176.468,20.808,153.145
C02587=1089.901,233.809,-75.857,176.465,20.806,153.145
C02588=1089.896,233.560,-75.831,176.462,20.804,153.145
C02589=1089.890,233.311,-75.805,176.460,20.802,153.145
C02590=1089.884,233.062,-75.779,176.456,20.800,153.145
C02591=1089.878,232.814,-75.753,176.453,20.797,153.145
C02592=1089.873,232.565,-75.728,176.451,20.795,153.145
C02593=1089.868,232.316,-75.702,176.448,20.792,153.145
C02594=1089.862,232.067,-75.676,176.446,20.790,153.145
C02595=1089.856,231.819,-75.650,176.442,20.788,153.145
C02596=1089.851,231.571,-75.624,176.439,20.785,153.145
C02597=1089.846,231.322,-75.598,176.437,20.783,153.145
C02598=1089.840,231.073,-75.572,176.434,20.781,153.145
C02599=1089.834,230.824,-75.547,176.431,20.779,153.145
C02600=1089.829,230.576,-75.522,176.428,20.776,153.145
C02601=1089.824,230.327,-75.496,176.426,20.774,153.145
C02602=1089.817,230.079,-75.470,176.423,20.772,153.145
C02603=1089.812,229.830,-75.444,176.419,20.769,153.145
C02604=1089.805,229.581,-75.418,176.417,20.767,153.145
C02605=1089.800,229.333,-75.393,176.414,20.765,153.145
C02606=1089.794,229.084,-75.367,176.411,20.763,153.145
C02607=1089.789,228.835,-75.341,176.408,20.760,153.145
C02608=1089.783,228.587,-75.316,176.406,20.758,153.145
C02609=1089.778,228.339,-75.291,176.403,20.756,153.145
C02610=1089.772,228.090,-75.265,176.399,20.754,153.145
C02611=1089.766,227.841,-75.239,176.397,20.752,153.145
C02612=1089.761,227.592,-75.213,176.394,20.749,153.145
C02613=1089.755,227.344,-75.188,176.392,20.747,153.144
C02614=1089.749,227.095,-75.162,176.388,20.744,153.144
C02615=1089.743,226.846,-75.137,176.386,20.742,153.144
C02616=1089.738,226.598,-75.112,176.383,20.740,153.144
C02617=1089.732,226.349,-75.086,176.381,20.738,153.144
C02618=1089.727,226.100,-75.060,176.377,20.735,153.144
C02619=1089.721,225.852,-75.036,176.374,20.733,153.144
C02620=1089.716,225.603,-75.010,176.372,20.731,153.144
C02621=1089.710,225.354,-74.985,176.369,20.729,153.144
C02622=1089.705,225.106,-74.959,176.366,20.727,153.144
C02623=1089.699,224.857,-74.934,176.363,20.724,153.144
C02624=1089.693,224.608,-74.908,176.361,20.722,153.144
C02625=1089.688,224.360,-74.883,176.358,20.719,153.144
C02626=1089.682,224.111,-74.858,176.355,20.717,153.144
C02627=1089.676,223.862,-74.832,176.352,20.715,153.144
C02628=1089.671,223.614,-74.807,176.350,20.713,153.144
C02629=1089.665,223.365,-74.781,176.346,20.710,153.144
C02630=1089.656,222.979,-74.743,176.343,20.707,153.144
C02631=1089.648,222.594,-74.704,176.338,20.704,153.144
C02632=1089.639,222.208,-74.664,176.334,20.700,153.144
C02633=1089.630,221.822,-74.626,176.329,20.696,153.144
C02634=1089.625,221.573,-74.600,176.327,20.694,153.144
C02635=1089.619,221.325,-74.575,176.324,20.692,153.144
C02636=1089.613,221.076,-74.550,176.321,20.690,153.144
C02637=1089.608,220.827,-74.524,176.318,20.687,153.144
C02638=1089.603,220.578,-74.500,176.316,20.685,153.144
C02639=1089.596,220.330,-74.475,176.312,20.683,153.144
C02640=1089.591,220.082,-74.450,176.310,20.681,153.144
C02641=1089.585,219.833,-74.425,176.307,20.679,153.144
C02642=1089.580,219.584,-74.400,176.304,20.677,153.143
C02643=1089.574,219.335,-74.375,176.301,20.674,153.143
C02644=1089.568,219.086,-74.350,176.299,20.672,153.143
C02645=1089.563,218.838,-74.325,176.296,20.670,153.143
C02646=1089.557,218.589,-74.299,176.293,20.668,153.143
C02647=1089.552,218.341,-74.274,176.290,20.665,153.143
C02648=1089.546,218.091,-74.250,176.288,20.663,153.143
C02649=1089.540,217.843,-74.226,176.285,20.661,153.143
C02650=1089.534,217.594,-74.200,176.282,20.659,153.143
C02651=1089.529,217.346,-74.176,176.279,20.656,153.143
C02652=1089.523,217.097,-74.150,176.277,20.654,153.143
C02653=1089.518,216.848,-74.126,176.274,20.652,153.143
C02654=1089.512,216.599,-74.100,176.271,20.650,153.143
C02655=1089.507,216.351,-74.076,176.268,20.647,153.143
C02656=1089.500,216.102,-74.051,176.266,20.645,153.143
C02657=1089.495,215.854,-74.027,176.263,20.643,153.143
C02658=1089.490,215.604,-74.001,176.260,20.641,153.143
C02659=1089.484,215.356,-73.976,176.257,20.638,153.143
C02660=1089.478,215.107,-73.952,176.255,20.636,153.143
C02661=1089.473,214.858,-73.928,176.251,20.634,153.143
C02662=1089.468,214.610,-73.903,176.249,20.632,153.143
C02663=1089.462,214.361,-73.878,176.246,20.630,153.143
C02664=1089.456,214.112,-73.854,176.244,20.627,153.143
C02665=1089.450,213.864,-73.828,176.241,20.625,153.143
C02666=1089.446,213.615,-73.804,176.238,20.623,153.143
C02667=1089.440,213.366,-73.779,176.235,20.620,153.143
C02668=1089.434,213.117,-73.755,176.233,20.618,153.143
C02669=1089.429,212.869,-73.730,176.229,20.616,153.143
C02670=1089.423,212.620,-73.705,176.227,20.614,153.143
C02671=1089.418,212.371,-73.681,176.224,20.611,153.143
C02672=1089.412,212.122,-73.656,176.221,20.609,153.143
C02673=1089.406,211.874,-73.631,176.219,20.607,153.143
C02674=1089.401,211.625,-73.607,176.216,20.605,153.143
C02675=1089.395,211.376,-73.582,176.214,20.603,153.142
C02676=1089.390,211.127,-73.558,176.210,20.601,153.142
C02677=1089.383,210.878,-73.534,176.208,20.599,153.142
C02678=1089.378,210.630,-73.510,176.205,20.596,153.142
C02679=1089.372,210.381,-73.486,176.202,20.594,153.142
C02680=1089.366,210.132,-73.460,176.199,20.592,153.142
C02681=1089.361,209.884,-73.436,176.197,20.590,153.142
C02682=1089.352,209.502,-73.398,176.193,20.586,153.142
C02683=1089.344,209.120,-73.362,176.188,20.582,153.142
C02684=1089.335,208.738,-73.324,176.184,20.579,153.142
C02685=1089.326,208.356,-73.286,176.180,20.576,153.142
C02686=1089.303,207.333,-73.188,176.110,20.541,153.146
C02687=1089.298,207.084,-73.164,176.107,20.540,153.146
C02688=1089.293,206.836,-73.140,176.104,20.539,153.147
C02689=1089.287,206.587,-73.116,176.101,20.537,153.147
C02690=1089.282,206.338,-73.093,176.098,20.536,153.147
C02691=1089.276,206.089,-73.068,176.096,20.534,153.147
C02692=1089.270,205.841,-73.045,176.093,20.533,153.147
C02693=1089.265,205.591,-73.021,176.090,20.532,153.147
C02694=1089.259,205.343,-72.997,176.088,20.531,153.148
C02695=1089.253,205.094,-72.973,176.084,20.529,153.148
C02696=1089.248,204.845,-72.950,176.081,20.528,153.148
C02697=1089.242,204.596,-72.925,176.078,20.527,153.148
C02698=1089.236,204.348,-72.901,176.076,20.525,153.148
C02699=1089.231,204.099,-72.878,176.073,20.524,153.149
C02700=1089.225,203.850,-72.854,176.071,20.523,153.149
C02701=1089.220,203.601,-72.830,176.067,20.521,153.149
C02702=1089.214,203.353,-72.807,176.064,20.520,153.149
C02703=1089.209,203.104,-72.783,176.062,20.518,153.149
C02704=1089.203,202.855,-72.760,176.059,20.517,153.150
C02705=1089.198,202.605,-72.736,176.056,20.516,153.150
C02706=1089.192,202.357,-72.712,176.054,20.515,153.150
C02707=1089.187,202.108,-72.689,176.050,20.513,153.150
C02708=1089.181,201.860,-72.665,176.047,20.512,153.150
C02709=1089.175,201.611,-72.642,176.045,20.511,153.151
C02710=1089.170,201.362,-72.618,176.042,20.510,153.151
C02711=1089.164,201.113,-72.595,176.039,20.509,153.151
C02712=1089.158,200.864,-72.570,176.036,20.508,153.151
C02713=1089.152,200.615,-72.547,176.034,20.506,153.151
C02714=1089.146,200.367,-72.523,176.030,20.505,153.152
C02715=1089.141,200.118,-72.500,176.028,20.503,153.152
C02716=1089.135,199.869,-72.477,176.025,20.502,153.152
C02717=1089.129,199.620,-72.453,176.022,20.501,153.152
C02718=1089.124,199.371,-72.430,176.019,20.500,153.152
C02719=1089.118,199.123,-72.406,176.017,20.499,153.153
C02720=1089.113,198.874,-72.383,176.014,20.497,153.153
C02721=1089.107,198.624,-72.359,176.011,20.496,153.153
C02722=1089.101,198.376,-72.336,176.008,20.494,153.153
C02723=1089.095,198.127,-72.313,176.005,20.493,153.153
C02724=1089.090,197.878,-72.289,176.003,20.492,153.153
C02725=1089.084,197.629,-72.265,176.000,20.491,153.154
C02726=1089.079,197.381,-72.243,175.997,20.489,153.154
C02727=1089.073,197.132,-72.220,175.994,20.488,153.154
C02728=1089.068,196.882,-72.196,175.992,20.487,153.154
C02729=1089.062,196.634,-72.172,175.989,20.486,153.154
C02730=1089.056,196.385,-72.149,175.986,20.484,153.154
C02731=1089.051,196.136,-72.126,175.983,20.483,153.155
C02732=1089.045,195.887,-72.103,175.980,20.481,153.155
C02733=1089.039,195.639,-72.079,175.977,20.480,153.155
C02734=1089.034,195.390,-72.056,175.975,20.479,153.155
C02735=1089.029,195.141,-72.033,175.972,20.478,153.155
C02736=1089.023,194.892,-72.010,175.969,20.477,153.156
C02737=1089.017,194.643,-71.987,175.967,20.476,153.156
C02738=1089.011,194.394,-71.964,175.964,20.474,153.156
C02739=1089.006,194.145,-71.940,175.962,20.473,153.156
C02740=1089.000,193.897,-71.917,175.959,20.472,153.156
C02741=1088.995,193.648,-71.894,175.956,20.470,153.156
C02742=1088.989,193.399,-71.871,175.953,20.469,153.157
C02743=1088.984,193.150,-71.847,175.950,20.467,153.157
C02744=1088.978,192.901,-71.824,175.947,20.466,153.157
C02745=1088.973,192.652,-71.802,175.945,20.465,153.157
C02746=1088.967,192.404,-71.779,175.942,20.463,153.157
C02747=1088.960,192.126,-71.753,175.939,20.462,153.158
C02748=1088.955,191.849,-71.727,175.936,20.460,153.158
C02749=1088.949,191.572,-71.702,175.933,20.459,153.158
C02750=1088.942,191.295,-71.675,175.930,20.457,153.158
C02751=1088.936,191.046,-71.653,175.927,20.456,153.158
C02752=1088.931,190.797,-71.630,175.924,20.455,153.158
C02753=1088.926,190.549,-71.606,175.922,20.453,153.159
C02754=1088.921,190.300,-71.583,175.919,20.452,153.159
C02755=1088.915,190.051,-71.561,175.916,20.451,153.159
C02756=1088.909,189.802,-71.538,175.914,20.450,153.159
C02757=1088.903,189.553,-71.515,175.911,20.449,153.159
C02758=1088.898,189.304,-71.492,175.908,20.447,153.159
C02759=1088.893,189.054,-71.469,175.906,20.446,153.160
C02760=1088.888,188.806,-71.446,175.903,20.445,153.160
C02761=1088.882,188.557,-71.423,175.900,20.443,153.160
C02762=1088.876,188.308,-71.400,175.898,20.442,153.160
C02763=1088.871,188.059,-71.377,175.895,20.441,153.160
C02764=1088.865,187.811,-71.355,175.892,20.439,153.160
C02765=1088.860,187.562,-71.332,175.890,20.438,153.161
C02766=1088.855,187.313,-71.308,175.886,20.436,153.161
C02767=1088.849,187.064,-71.286,175.884,20.435,153.161
C02768=1088.844,186.815,-71.263,175.881,20.433,153.161
C02769=1088.838,186.566,-71.240,175.878,20.432,153.161
C02770=1088.833,186.318,-71.218,175.876,20.431,153.161
C02771=1088.827,186.069,-71.195,175.873,20.429,153.162
C02772=1088.822,185.819,-71.173,175.871,20.428,153.162
C02773=1088.816,185.570,-71.150,175.868,20.427,153.162
C02774=1088.811,185.322,-71.127,175.865,20.425,153.162
C02775=1088.805,185.073,-71.104,175.863,20.424,153.162
C02776=1088.800,184.824,-71.082,175.860,20.423,153.162
C02777=1088.794,184.575,-71.059,175.857,20.422,153.162
C02778=1088.788,184.326,-71.036,175.854,20.421,153.163
C02779=1088.783,184.076,-71.014,175.852,20.419,153.163
C02780=1088.776,183.828,-70.991,175.849,20.418,153.163
C02781=1088.771,183.580,-70.969,175.847,20.417,153.163
C02782=1088.766,183.330,-70.947,175.844,20.416,153.163
C02783=1088.760,183.081,-70.924,175.841,20.414,153.164
C02784=1088.754,182.833,-70.901,175.838,20.413,153.164
C02785=1088.748,182.583,-70.879,175.836,20.412,153.164
C02786=1088.742,182.334,-70.856,175.833,20.410,153.164
C02787=1088.737,182.086,-70.834,175.830,20.409,153.164
C02788=1088.731,181.837,-70.812,175.828,20.408,153.164
C02789=1088.725,181.588,-70.789,175.825,20.407,153.165
C02790=1088.720,181.338,-70.767,175.823,20.405,153.165
C02791=1088.713,181.090,-70.744,175.820,20.404,153.165
C02792=1088.708,180.841,-70.721,175.817,20.403,153.165
C02793=1088.703,180.592,-70.700,175.815,20.401,153.165
C02794=1088.696,180.344,-70.677,175.812,20.400,153.166
C02795=1088.691,180.094,-70.655,175.809,20.399,153.166
C02796=1088.685,179.845,-70.632,175.806,20.398,153.166
C02797=1088.680,179.596,-70.610,175.804,20.396,153.166
C02798=1088.674,179.348,-70.588,175.801,20.395,153.166
C02799=1088.669,179.098,-70.566,175.798,20.394,153.166
C02800=1088.663,178.849,-70.543,175.796,20.393,153.167
C02801=1088.657,178.601,-70.521,175.793,20.391,153.167
C02802=1088.652,178.352,-70.498,175.791,20.390,153.167
C02803=1088.646,178.102,-70.476,175.788,20.389,153.167
C02804=1088.640,177.854,-70.454,175.785,20.387,153.167
C02805=1088.635,177.605,-70.432,175.783,20.386,153.167
C02806=1088.629,177.356,-70.410,175.780,20.385,153.168
C02807=1088.623,177.107,-70.387,175.777,20.383,153.168
C02808=1088.618,176.858,-70.365,175.775,20.382,153.168
C02809=1088.612,176.609,-70.343,175.772,20.381,153.168
C02810=1088.606,176.360,-70.321,175.770,20.379,153.168
C02811=1088.601,176.082,-70.296,175.767,20.378,153.168
C02812=1088.594,175.806,-70.272,175.764,20.377,153.168
C02813=1088.588,175.527,-70.247,175.761,20.375,153.169
C02814=1088.582,175.250,-70.222,175.758,20.374,153.169
C02815=1088.576,175.002,-70.201,175.755,20.372,153.169
C02816=1088.571,174.752,-70.178,175.753,20.371,153.169
C02817=1088.564,174.504,-70.156,175.750,20.369,153.169
C02818=1088.559,174.255,-70.134,175.747,20.369,153.170
C02819=1088.554,174.005,-70.112,175.745,20.367,153.170
C02820=1088.548,173.756,-70.090,175.742,20.366,153.170
C02821=1088.543,173.508,-70.068,175.740,20.364,153.170
C02822=1088.536,173.259,-70.046,175.737,20.363,153.170
C02823=1088.532,173.010,-70.024,175.734,20.362,153.170
C02824=1088.525,172.761,-70.003,175.733,20.361,153.170
C02825=1088.520,172.512,-69.980,175.730,20.359,153.170
C02826=1088.515,172.263,-69.958,175.727,20.358,153.171
C02827=1088.509,172.014,-69.936,175.725,20.357,153.171
C02828=1088.504,171.765,-69.914,175.722,20.355,153.171
C02829=1088.498,171.516,-69.893,175.720,20.354,153.171
C02830=1088.492,171.266,-69.870,175.717,20.352,153.171
C02831=1088.486,171.018,-69.849,175.714,20.351,153.171
C02832=1088.481,170.769,-69.826,175.712,20.350,153.172
C02833=1088.475,170.520,-69.805,175.709,20.348,153.172
C02834=1088.470,170.271,-69.783,175.706,20.347,153.172
C02835=1088.464,170.022,-69.762,175.704,20.345,153.172
C02836=1088.459,169.773,-69.739,175.701,20.344,153.172
C02837=1088.453,169.524,-69.718,175.699,20.342,153.172
C02838=1088.448,169.275,-69.696,175.696,20.341,153.172
C02839=1088.443,169.026,-69.674,175.693,20.340,153.173
C02840=1088.437,168.777,-69.652,175.692,20.339,153.173
C02841=1088.432,168.528,-69.630,175.689,20.338,153.173
C02842=1088.426,168.279,-69.609,175.687,20.336,153.173
C02843=1088.420,168.030,-69.588,175.684,20.335,153.173
C02844=1088.415,167.781,-69.565,175.681,20.333,153.173
C02845=1088.409,167.532,-69.544,175.679,20.332,153.173
C02846=1088.404,167.283,-69.522,175.676,20.330,153.173
C02847=1088.398,167.034,-69.501,175.674,20.329,153.173
C02848=1088.393,166.785,-69.478,175.671,20.327,153.174
C02849=1088.387,166.536,-69.457,175.669,20.326,153.174
C02850=1088.382,166.287,-69.435,175.666,20.324,153.174
C02851=1088.376,166.038,-69.414,175.663,20.323,153.174
C02852=1088.372,165.789,-69.392,175.661,20.322,153.174
C02853=1088.366,165.540,-69.370,175.659,20.321,153.174
C02854=1088.361,165.291,-69.348,175.656,20.319,153.174
C02855=1088.355,165.042,-69.327,175.654,20.318,153.174
C02856=1088.349,164.793,-69.305,175.651,20.316,153.175
C02857=1088.344,164.544,-69.283,175.649,20.315,153.175
C02858=1088.338,164.295,-69.262,175.646,20.314,153.175
C02859=1088.333,164.046,-69.241,175.644,20.312,153.175
C02860=1088.327,163.797,-69.219,175.641,20.311,153.175
C02861=1088.322,163.548,-69.197,175.638,20.309,153.175
C02862=1088.316,163.299,-69.175,175.637,20.308,153.175
C02863=1088.311,163.050,-69.155,175.634,20.307,153.175
C02864=1088.306,162.801,-69.133,175.632,20.305,153.176
C02865=1088.300,162.552,-69.111,175.629,20.304,153.176
C02866=1088.295,162.303,-69.090,175.626,20.302,153.176
C02867=1088.290,162.054,-69.068,175.624,20.301,153.176
C02868=1088.284,161.805,-69.047,175.621,20.299,153.176
C02869=1088.279,161.556,-69.025,175.619,20.297,153.176
C02870=1088.273,161.307,-69.004,175.616,20.296,153.176
C02871=1088.267,161.058,-68.983,175.614,20.295,153.176
C02872=1088.262,160.809,-68.962,175.612,20.294,153.176
C02873=1088.256,160.560,-68.940,175.609,20.292,153.177
C02874=1088.250,160.311,-68.919,175.607,20.291,153.177
C02875=1088.245,160.033,-68.895,175.604,20.289,153.177
C02876=1088.238,159.755,-68.871,175.602,20.288,153.177
C02877=1088.232,159.477,-68.848,175.598,20.286,153.177
C02878=1088.225,159.199,-68.824,175.596,20.285,153.177
C02879=1088.220,158.951,-68.803,175.593,20.283,153.177
C02880=1088.214,158.701,-68.782,175.590,20.282,153.177
C02881=1088.209,158.452,-68.760,175.589,20.281,153.178
C02882=1088.204,158.203,-68.740,175.586,20.279,153.178
C02883=1088.198,157.954,-68.718,175.584,20.278,153.178
C02884=1088.192,157.706,-68.697,175.581,20.276,153.178
C02885=1088.187,157.456,-68.676,175.578,20.275,153.178
C02886=1088.181,157.207,-68.655,175.576,20.273,153.178
C02887=1088.175,156.958,-68.634,175.573,20.272,153.178
C02888=1088.170,156.710,-68.613,175.572,20.271,153.178
C02889=1088.164,156.460,-68.592,175.569,20.269,153.178
C02890=1088.158,156.211,-68.571,175.566,20.268,153.179
C02891=1088.153,155.962,-68.550,175.564,20.266,153.179
C02892=1088.148,155.713,-68.528,175.561,20.265,153.179
C02893=1088.143,155.463,-68.507,175.559,20.263,153.179
C02894=1088.137,155.215,-68.486,175.556,20.262,153.179
C02895=1088.130,154.965,-68.466,175.554,20.261,153.179
C02896=1088.125,154.717,-68.444,175.552,20.260,153.179
C02897=1088.120,154.468,-68.424,175.549,20.258,153.179
C02898=1088.113,154.219,-68.402,175.547,20.257,153.180
C02899=1088.108,153.969,-68.382,175.544,20.255,153.180
C02900=1088.103,153.721,-68.360,175.542,20.254,153.180
C02901=1088.097,153.471,-68.339,175.540,20.253,153.180
C02902=1088.091,153.223,-68.318,175.537,20.251,153.180
C02903=1088.086,152.974,-68.298,175.535,20.250,153.180
C02904=1088.080,152.724,-68.277,175.532,20.248,153.180
C02905=1088.074,152.475,-68.255,175.530,20.247,153.180
C02906=1088.069,152.226,-68.235,175.527,20.245,153.180
C02907=1088.064,151.977,-68.214,175.525,20.244,153.181
C02908=1088.058,151.728,-68.193,175.523,20.243,153.181
C02909=1088.053,151.479,-68.172,175.520,20.241,153.181
C02910=1088.047,151.229,-68.152,175.518,20.239,153.181
C02911=1088.042,150.981,-68.130,175.515,20.238,153.181
C02912=1088.035,150.731,-68.110,175.513,20.236,153.181
C02913=1088.030,150.482,-68.089,175.511,20.235,153.181
C02914=1088.024,150.234,-68.068,175.508,20.234,153.181
C02915=1088.019,149.985,-68.048,175.506,20.233,153.181
C02916=1088.014,149.736,-68.027,175.503,20.231,153.181
C02917=1088.008,149.486,-68.006,175.501,20.230,153.182
C02918=1088.002,149.237,-67.985,175.499,20.229,153.182
C02919=1087.997,148.988,-67.964,175.497,20.227,153.182
C02920=1087.991,148.739,-67.944,175.494,20.225,153.182
C02921=1087.985,148.489,-67.923,175.492,20.224,153.182
C02922=1087.980,148.241,-67.902,175.489,20.222,153.182
C02923=1087.974,147.992,-67.882,175.487,20.221,153.182
C02924=1087.968,147.743,-67.862,175.485,20.220,153.182
C02925=1087.963,147.494,-67.841,175.482,20.218,153.182
C02926=1087.957,147.244,-67.820,175.480,20.217,153.182
C02927=1087.952,146.995,-67.800,175.477,20.215,153.183
C02928=1087.946,146.747,-67.779,175.475,20.214,153.183
C02929=1087.941,146.498,-67.758,175.473,20.212,153.183
C02930=1087.935,146.249,-67.738,175.470,20.211,153.183
C02931=1087.929,145.999,-67.717,175.468,20.209,153.183
C02932=1087.923,145.750,-67.697,175.465,20.208,153.183
C02933=1087.918,145.501,-67.676,175.464,20.207,153.183
C02934=1087.913,145.252,-67.656,175.461,20.205,153.183
C02935=1087.907,145.003,-67.636,175.459,20.204,153.183
C02936=1087.901,144.753,-67.615,175.456,20.202,153.183
C02937=1087.896,144.505,-67.594,175.453,20.201,153.183
C02938=1087.890,144.256,-67.574,175.452,20.200,153.184
C02939=1087.884,143.977,-67.551,175.449,20.198,153.184
C02940=1087.878,143.699,-67.528,175.446,20.196,153.184
C02941=1087.871,143.421,-67.505,175.443,20.194,153.184
C02942=1087.865,143.143,-67.483,175.441,20.193,153.184
C02943=1087.859,142.894,-67.462,175.438,20.191,153.184
C02944=1087.854,142.645,-67.441,175.437,20.190,153.184
C02945=1087.848,142.396,-67.421,175.434,20.188,153.184
C02946=1087.843,142.147,-67.401,175.432,20.187,153.184
C02947=1087.838,141.898,-67.380,175.429,20.185,153.184
C02948=1087.831,141.648,-67.361,175.427,20.184,153.184
C02949=1087.826,141.399,-67.340,175.425,20.182,153.184
C02950=1087.820,141.150,-67.320,175.422,20.181,153.185
C02951=1087.815,140.901,-67.300,175.420,20.179,153.185
C02952=1087.810,140.652,-67.279,175.418,20.178,153.185
C02953=1087.804,140.403,-67.259,175.416,20.176,153.185
C02954=1087.798,140.154,-67.239,175.413,20.175,153.185
C02955=1087.792,139.905,-67.219,175.411,20.174,153.185
C02956=1087.787,139.656,-67.198,175.408,20.172,153.185
C02957=1087.781,139.407,-67.178,175.407,20.171,153.185
C02958=1087.776,139.157,-67.158,175.404,20.169,153.185
C02959=1087.770,138.909,-67.138,175.402,20.168,153.185
C02960=1087.764,138.659,-67.117,175.399,20.166,153.185
C02961=1087.758,138.410,-67.097,175.397,20.165,153.185
C02962=1087.753,138.161,-67.077,175.395,20.163,153.186
C02963=1087.747,137.912,-67.057,175.392,20.162,153.186
C02964=1087.742,137.662,-67.037,175.390,20.160,153.186
C02965=1087.736,137.413,-67.017,175.388,20.159,153.186
C02966=1087.731,137.164,-66.997,175.386,20.157,153.186
C02967=1087.725,136.916,-66.977,175.383,20.156,153.186
C02968=1087.720,136.666,-66.957,175.381,20.154,153.186
C02969=1087.714,136.417,-66.937,175.379,20.153,153.186
C02970=1087.708,136.168,-66.917,175.377,20.151,153.186
C02971=1087.703,135.919,-66.896,175.374,20.149,153.186
C02972=1087.697,135.670,-66.877,175.372,20.148,153.186
C02973=1087.692,135.420,-66.857,175.370,20.147,153.186
C02974=1087.686,135.172,-66.837,175.368,20.145,153.186
C02975=1087.681,134.922,-66.817,175.365,20.144,153.187
C02976=1087.675,134.673,-66.797,175.363,20.143,153.187
C02977=1087.669,134.424,-66.777,175.361,20.141,153.187
C02978=1087.664,134.175,-66.757,175.358,20.139,153.187
C02979=1087.658,133.926,-66.737,175.356,20.138,153.187
C02980=1087.653,133.677,-66.716,175.354,20.136,153.187
C02981=1087.647,133.427,-66.697,175.352,20.135,153.187
C02982=1087.641,133.178,-66.677,175.349,20.133,153.187
C02983=1087.636,132.929,-66.657,175.347,20.131,153.187
C02984=1087.630,132.680,-66.637,175.345,20.130,153.187
C02985=1087.624,132.431,-66.617,175.343,20.128,153.187
C02986=1087.619,132.181,-66.598,175.340,20.127,153.187
C02987=1087.613,131.932,-66.578,175.339,20.126,153.187
C02988=1087.607,131.683,-66.558,175.336,20.124,153.187
C02989=1087.601,131.434,-66.538,175.334,20.122,153.187
C02990=1087.596,131.185,-66.518,175.331,20.121,153.188
C02991=1087.590,130.936,-66.499,175.330,20.119,153.187
C02992=1087.584,130.687,-66.479,175.327,20.118,153.188
C02993=1087.579,130.437,-66.459,175.324,20.116,153.188
C02994=1087.573,130.189,-66.440,175.323,20.115,153.188
C02995=1087.567,129.939,-66.420,175.320,20.113,153.188
C02996=1087.562,129.690,-66.400,175.318,20.112,153.188
C02997=1087.556,129.441,-66.380,175.316,20.110,153.188
C02998=1087.550,129.192,-66.361,175.314,20.109,153.188
C02999=1087.544,128.942,-66.341,175.311,20.108,153.188
C03000=1087.539,128.693,-66.322,175.309,20.106,153.188
C03001=1087.533,128.444,-66.302,175.307,20.105,153.188
C03002=1087.528,128.195,-66.283,175.305,20.103,153.188
C03003=1087.522,127.917,-66.261,175.302,20.101,153.188
C03004=1087.515,127.638,-66.239,175.300,20.099,153.188
C03005=1087.508,127.361,-66.216,175.297,20.098,153.188
C03006=1087.502,127.083,-66.195,175.295,20.096,153.189
C03007=1087.496,126.833,-66.175,175.292,20.094,153.189
C03008=1087.491,126.584,-66.157,175.290,20.093,153.189
C03009=1087.485,126.336,-66.137,175.288,20.091,153.189
C03010=1087.479,126.086,-66.117,175.286,20.090,153.189
C03011=1087.474,125.837,-66.098,175.284,20.088,153.189
C03012=1087.468,125.588,-66.078,175.282,20.087,153.189
C03013=1087.463,125.338,-66.058,175.279,20.085,153.189
C03014=1087.457,125.089,-66.039,175.277,20.083,153.189
C03015=1087.451,124.840,-66.019,175.275,20.082,153.189
C03016=1087.446,124.591,-66.000,175.273,20.080,153.189
C03017=1087.440,124.342,-65.981,175.271,20.079,153.189
C03018=1087.435,124.092,-65.962,175.269,20.078,153.189
C03019=1087.429,123.843,-65.942,175.267,20.076,153.189
C03020=1087.423,123.594,-65.923,175.264,20.074,153.189
C03021=1087.417,123.345,-65.903,175.262,20.072,153.189
C03022=1087.412,123.095,-65.884,175.260,20.071,153.189
C03023=1087.406,122.847,-65.864,175.258,20.069,153.189
C03024=1087.400,122.598,-65.845,175.255,20.068,153.189
C03025=1087.395,122.348,-65.826,175.254,20.066,153.189
C03026=1087.390,122.098,-65.806,175.251,20.065,153.189
C03027=1087.384,121.850,-65.786,175.249,20.063,153.189
C03028=1087.379,121.601,-65.767,175.247,20.062,153.190
C03029=1087.373,121.351,-65.748,175.245,20.060,153.190
C03030=1087.367,121.102,-65.729,175.242,20.058,153.190
C03031=1087.362,120.853,-65.710,175.241,20.057,153.190
C03032=1087.356,120.603,-65.690,175.238,20.055,153.190
C03033=1087.351,120.354,-65.671,175.236,20.053,153.190
C03034=1087.345,120.106,-65.651,175.234,20.052,153.190
C03035=1087.339,119.856,-65.632,175.232,20.050,153.190
C03036=1087.334,119.607,-65.613,175.229,20.048,153.190
C03037=1087.328,119.358,-65.594,175.228,20.047,153.190
C03038=1087.323,119.109,-65.575,175.225,20.045,153.190
C03039=1087.317,118.859,-65.556,175.223,20.043,153.190
C03040=1087.311,118.610,-65.536,175.221,20.042,153.190
C03041=1087.306,118.361,-65.517,175.219,20.041,153.190
C03042=1087.301,118.112,-65.498,175.216,20.039,153.190
C03043=1087.295,117.862,-65.479,175.215,20.037,153.190
C03044=1087.290,117.613,-65.460,175.212,20.036,153.190
C03045=1087.284,117.364,-65.441,175.210,20.034,153.190
C03046=1087.278,117.115,-65.422,175.209,20.032,153.190
C03047=1087.273,116.866,-65.403,175.206,20.031,153.190
C03048=1087.267,116.617,-65.384,175.204,20.029,153.190
C03049=1087.261,116.367,-65.365,175.202,20.027,153.190
C03050=1087.256,116.118,-65.346,175.200,20.025,153.190
C03051=1087.250,115.869,-65.327,175.197,20.024,153.190
C03052=1087.245,115.620,-65.308,175.196,20.022,153.190
C03053=1087.239,115.370,-65.288,175.194,20.020,153.190
C03054=1087.234,115.121,-65.269,175.192,20.019,153.190
C03055=1087.228,114.872,-65.250,175.189,20.017,153.190
C03056=1087.223,114.623,-65.231,175.187,20.015,153.190
C03057=1087.218,114.374,-65.212,175.186,20.014,153.190
C03058=1087.212,114.124,-65.193,175.183,20.012,153.190
C03059=1087.205,113.875,-65.174,175.181,20.010,153.190
C03060=1087.201,113.626,-65.156,175.179,20.009,153.190
C03061=1087.195,113.377,-65.137,175.177,20.007,153.190
C03062=1087.189,113.127,-65.117,175.174,20.005,153.190
C03063=1087.183,112.879,-65.099,175.173,20.004,153.190
C03064=1087.178,112.629,-65.080,175.170,20.002,153.190
C03065=1087.172,112.380,-65.061,175.168,20.000,153.190
C03066=1087.167,112.131,-65.042,175.167,19.999,153.190
C03067=1087.160,111.853,-65.021,175.164,19.997,153.190
C03068=1087.154,111.574,-65.001,175.162,19.996,153.190
C03069=1087.148,111.296,-64.979,175.159,19.994,153.190
C03070=1087.141,111.018,-64.959,175.157,19.992,153.190
C03071=1087.136,110.769,-64.939,175.155,19.990,153.190
C03072=1087.130,110.519,-64.920,175.153,19.989,153.190
C03073=1087.125,110.270,-64.903,175.151,19.987,153.190
C03074=1087.119,110.021,-64.883,175.149,19.985,153.190
C03075=1087.112,109.772,-64.865,175.147,19.984,153.191
C03076=1087.107,109.523,-64.846,175.144,19.982,153.191
C03077=1087.102,109.273,-64.827,175.143,19.980,153.190
C03078=1087.096,109.024,-64.809,175.140,19.978,153.190
C03079=1087.090,108.775,-64.790,175.139,19.977,153.191
C03080=1087.085,108.526,-64.771,175.136,19.975,153.191
C03081=1087.079,108.277,-64.753,175.134,19.973,153.191
C03082=1087.074,108.027,-64.734,175.132,19.972,153.191
C03083=1087.067,107.778,-64.715,175.130,19.970,153.191
C03084=1087.062,107.529,-64.697,175.128,19.968,153.191
C03085=1087.057,107.279,-64.678,175.126,19.967,153.191
C03086=1087.051,107.031,-64.659,175.124,19.965,153.191
C03087=1087.045,106.781,-64.641,175.122,19.964,153.191
C03088=1087.039,106.532,-64.622,175.120,19.962,153.191
C03089=1087.034,106.282,-64.604,175.117,19.960,153.191
C03090=1087.028,106.033,-64.585,175.116,19.958,153.191
C03091=1087.023,105.784,-64.567,175.114,19.956,153.191
C03092=1087.017,105.534,-64.548,175.112,19.955,153.191
C03093=1087.011,105.285,-64.529,175.110,19.953,153.191
C03094=1087.006,105.036,-64.511,175.107,19.951,153.191
C03095=1087.000,104.787,-64.493,175.106,19.950,153.191
C03096=1086.995,104.537,-64.474,175.103,19.948,153.191
C03097=1086.988,104.288,-64.456,175.102,19.947,153.191
C03098=1086.984,104.039,-64.438,175.099,19.945,153.191
C03099=1086.977,103.790,-64.419,175.097,19.943,153.191
C03100=1086.972,103.541,-64.400,175.096,19.942,153.191
C03101=1086.966,103.291,-64.382,175.093,19.940,153.191
C03102=1086.961,103.043,-64.363,175.092,19.938,153.191
C03103=1086.955,102.793,-64.345,175.090,19.936,153.191
C03104=1086.950,102.544,-64.327,175.087,19.934,153.191
C03105=1086.944,102.294,-64.308,175.085,19.933,153.191
C03106=1086.939,102.045,-64.290,175.083,19.931,153.191
C03107=1086.932,101.796,-64.272,175.082,19.930,153.191
C03108=1086.928,101.547,-64.254,175.079,19.928,153.191
C03109=1086.921,101.297,-64.235,175.077,19.926,153.191
C03110=1086.916,101.048,-64.217,175.076,19.924,153.191
C03111=1086.910,100.799,-64.198,175.073,19.922,153.190
C03112=1086.905,100.550,-64.180,175.072,19.921,153.190
C03113=1086.899,100.300,-64.162,175.069,19.919,153.191
C03114=1086.893,100.051,-64.144,175.068,19.918,153.191
C03115=1086.888,99.801,-64.125,175.065,19.916,153.191
C03116=1086.882,99.553,-64.107,175.063,19.914,153.191
C03117=1086.876,99.303,-64.089,175.062,19.912,153.190
C03118=1086.871,99.054,-64.071,175.059,19.910,153.190
C03119=1086.865,98.805,-64.052,175.058,19.909,153.190
C03120=1086.859,98.556,-64.035,175.055,19.907,153.191
C03121=1086.853,98.306,-64.017,175.053,19.905,153.191
C03122=1086.848,98.057,-63.998,175.051,19.904,153.190
C03123=1086.842,97.808,-63.980,175.049,19.902,153.190
C03124=1086.836,97.558,-63.962,175.048,19.900,153.190
C03125=1086.831,97.308,-63.944,175.045,19.898,153.190
C03126=1086.825,97.060,-63.925,175.044,19.897,153.190
C03127=1086.819,96.810,-63.907,175.041,19.895,153.190
C03128=1086.814,96.561,-63.889,175.039,19.893,153.190
C03129=1086.808,96.312,-63.871,175.038,19.891,153.190
C03130=1086.802,96.063,-63.853,175.035,19.889,153.190
C03131=1086.796,95.785,-63.833,175.033,19.887,153.190
C03132=1086.790,95.506,-63.814,175.031,19.886,153.190
C03133=1086.784,95.228,-63.793,175.029,19.884,153.190
C03134=1086.777,94.950,-63.772,175.027,19.882,153.190
C03135=1086.772,94.701,-63.755,175.024,19.880,153.190
C03136=1086.766,94.451,-63.737,175.023,19.879,153.190
C03137=1086.760,94.202,-63.719,175.021,19.877,153.190
C03138=1086.755,93.953,-63.700,175.019,19.875,153.190
C03139=1086.749,93.703,-63.682,175.017,19.873,153.190
C03140=1086.743,93.454,-63.665,175.015,19.872,153.190
C03141=1086.738,93.205,-63.647,175.013,19.870,153.190
C03142=1086.732,92.955,-63.629,175.011,19.868,153.190
C03143=1086.727,92.707,-63.611,175.009,19.866,153.190
C03144=1086.721,92.458,-63.593,175.007,19.864,153.190
C03145=1086.715,92.208,-63.575,175.005,19.863,153.190
C03146=1086.710,91.959,-63.557,175.003,19.861,153.190
C03147=1086.705,91.710,-63.539,175.002,19.859,153.190
C03148=1086.699,91.460,-63.521,174.999,19.857,153.190
C03149=1086.693,91.211,-63.504,174.998,19.856,153.190
C03150=1086.687,90.961,-63.486,174.996,19.854,153.190
C03151=1086.681,90.712,-63.468,174.993,19.852,153.190
C03152=1086.676,90.463,-63.451,174.992,19.850,153.190
C03153=1086.671,90.213,-63.432,174.989,19.848,153.190
C03154=1086.665,89.964,-63.415,174.988,19.847,153.190
C03155=1086.659,89.715,-63.397,174.986,19.845,153.190
C03156=1086.653,89.465,-63.379,174.984,19.843,153.190
C03157=1086.648,89.216,-63.362,174.982,19.841,153.190
C03158=1086.642,88.966,-63.344,174.980,19.840,153.190
C03159=1086.636,88.717,-63.326,174.978,19.838,153.190
C03160=1086.631,88.468,-63.308,174.977,19.836,153.190
C03161=1086.625,88.218,-63.291,174.974,19.834,153.190
C03162=1086.619,87.969,-63.273,174.972,19.832,153.190
C03163=1086.614,87.720,-63.255,174.970,19.831,153.189
C03164=1086.607,87.471,-63.237,174.968,19.829,153.189
C03165=1086.602,87.222,-63.220,174.967,19.827,153.189
C03166=1086.596,86.973,-63.202,174.964,19.825,153.189
C03167=1086.590,86.723,-63.184,174.963,19.824,153.189
C03168=1086.585,86.474,-63.167,174.961,19.821,153.189
C03169=1086.579,86.225,-63.149,174.959,19.820,153.189
C03170=1086.573,85.975,-63.131,174.957,19.818,153.189
C03171=1086.568,85.726,-63.114,174.955,19.816,153.189
C03172=1086.562,85.476,-63.097,174.953,19.814,153.189
C03173=1086.556,85.227,-63.079,174.952,19.813,153.189
C03174=1086.551,84.978,-63.061,174.949,19.811,153.189
C03175=1086.545,84.728,-63.044,174.948,19.809,153.189
C03176=1086.539,84.480,-63.027,174.946,19.807,153.189
C03177=1086.533,84.230,-63.009,174.944,19.806,153.189
C03178=1086.527,83.981,-62.991,174.942,19.804,153.189
C03179=1086.522,83.731,-62.975,174.940,19.802,153.189
C03180=1086.517,83.482,-62.957,174.938,19.800,153.189
C03181=1086.510,83.233,-62.939,174.936,19.798,153.189
C03182=1086.505,82.983,-62.921,174.934,19.796,153.189
C03183=1086.499,82.734,-62.904,174.932,19.794,153.189
C03184=1086.494,82.485,-62.887,174.931,19.793,153.189
C03185=1086.488,82.235,-62.869,174.928,19.791,153.189
C03186=1086.483,81.986,-62.852,174.927,19.789,153.188
C03187=1086.477,81.737,-62.834,174.925,19.787,153.188
C03188=1086.472,81.487,-62.817,174.923,19.786,153.188
C03189=1086.466,81.238,-62.799,174.921,19.784,153.188
C03190=1086.460,80.989,-62.782,174.919,19.782,153.188
C03191=1086.454,80.739,-62.765,174.917,19.780,153.188
C03192=1086.449,80.490,-62.748,174.916,19.778,153.188
C03193=1086.443,80.241,-62.730,174.914,19.776,153.188
C03194=1086.438,79.991,-62.713,174.912,19.775,153.188
C03195=1086.432,79.714,-62.693,174.910,19.773,153.188
C03196=1086.425,79.435,-62.674,174.908,19.770,153.188
C03197=1086.419,79.157,-62.655,174.905,19.768,153.188
C03198=1086.413,78.878,-62.636,174.904,19.766,153.188
C03199=1086.407,78.629,-62.618,174.902,19.764,153.188
C03200=1086.401,78.381,-62.601,174.900,19.763,153.188
C03201=1086.396,78.131,-62.584,174.898,19.761,153.188
C03202=1086.390,77.882,-62.567,174.896,19.759,153.188
C03203=1086.385,77.633,-62.549,174.894,19.757,153.188
C03204=1086.378,77.383,-62.532,174.893,19.755,153.187
C03205=1086.373,77.134,-62.515,174.891,19.753,153.187
C03206=1086.367,76.884,-62.498,174.889,19.752,153.187
C03207=1086.361,76.635,-62.481,174.887,19.750,153.187
C03208=1086.356,76.386,-62.464,174.885,19.748,153.187
C03209=1086.350,76.136,-62.446,174.883,19.746,153.187
C03210=1086.344,75.887,-62.429,174.882,19.744,153.187
C03211=1086.338,75.638,-62.412,174.879,19.742,153.187
C03212=1086.333,75.388,-62.395,174.878,19.741,153.187
C03213=1086.328,75.139,-62.378,174.876,19.739,153.187
C03214=1086.321,74.890,-62.361,174.874,19.737,153.187
C03215=1086.315,74.640,-62.344,174.872,19.735,153.187
C03216=1086.310,74.391,-62.326,174.871,19.733,153.187
C03217=1086.304,74.141,-62.310,174.868,19.731,153.187
C03218=1086.298,73.892,-62.292,174.867,19.729,153.187
C03219=1086.293,73.643,-62.276,174.865,19.727,153.187
C03220=1086.287,73.394,-62.259,174.863,19.726,153.187
C03221=1086.282,73.144,-62.242,174.861,19.724,153.187
C03222=1086.277,72.895,-62.225,174.860,19.722,153.186
C03223=1086.270,72.645,-62.208,174.857,19.720,153.186
C03224=1086.265,72.396,-62.191,174.856,19.718,153.186
C03225=1086.259,72.146,-62.173,174.854,19.716,153.186
C03226=1086.253,71.897,-62.157,174.852,19.714,153.186
C03227=1086.248,71.648,-62.139,174.850,19.712,153.186
C03228=1086.242,71.399,-62.123,174.849,19.711,153.186
C03229=1086.236,71.149,-62.106,174.846,19.709,153.186
C03230=1086.231,70.900,-62.089,174.845,19.707,153.186
C03231=1086.225,70.651,-62.072,174.843,19.705,153.186
C03232=1086.220,70.401,-62.056,174.841,19.703,153.186
C03233=1086.213,70.152,-62.039,174.839,19.701,153.186
C03234=1086.208,69.902,-62.021,174.838,19.699,153.186
C03235=1086.202,69.653,-62.005,174.836,19.698,153.186
C03236=1086.196,69.404,-61.988,174.834,19.695,153.186
C03237=1086.191,69.154,-61.971,174.833,19.694,153.185
C03238=1086.185,68.905,-61.954,174.830,19.692,153.185
C03239=1086.179,68.656,-61.937,174.829,19.690,153.185
C03240=1086.174,68.406,-61.921,174.827,19.688,153.185
C03241=1086.168,68.156,-61.904,174.825,19.686,153.185
C03242=1086.162,67.907,-61.888,174.823,19.684,153.185
C03243=1086.157,67.658,-61.870,174.822,19.682,153.185
C03244=1086.151,67.409,-61.854,174.819,19.680,153.185
C03245=1086.145,67.159,-61.837,174.818,19.679,153.185
C03246=1086.139,66.910,-61.820,174.816,19.677,153.185
C03247=1086.133,66.661,-61.804,174.814,19.675,153.185
C03248=1086.128,66.411,-61.787,174.812,19.673,153.185
C03249=1086.122,66.162,-61.770,174.811,19.671,153.185
C03250=1086.117,65.912,-61.754,174.809,19.669,153.185
C03251=1086.111,65.664,-61.737,174.807,19.667,153.185
C03252=1086.106,65.414,-61.720,174.806,19.666,153.185
C03253=1086.100,65.165,-61.704,174.804,19.663,153.184
C03254=1086.094,64.915,-61.687,174.802,19.662,153.184
C03255=1086.088,64.666,-61.670,174.800,19.660,153.184
C03256=1086.082,64.416,-61.654,174.799,19.658,153.184
C03257=1086.076,64.167,-61.636,174.796,19.656,153.184
C03258=1086.070,63.917,-61.620,174.795,19.654,153.184
C03259=1086.065,63.639,-61.602,174.793,19.652,153.184
C03260=1086.058,63.361,-61.583,174.790,19.650,153.184
C03261=1086.051,63.083,-61.565,174.789,19.648,153.184
C03262=1086.045,62.805,-61.547,174.787,19.646,153.184
C03263=1086.039,62.555,-61.531,174.785,19.644,153.184
C03264=1086.033,62.306,-61.514,174.783,19.642,153.184
C03265=1086.027,62.057,-61.497,174.782,19.640,153.184
C03266=1086.022,61.807,-61.481,174.779,19.638,153.184
C03267=1086.016,61.558,-61.464,174.778,19.637,153.183
C03268=1086.010,61.309,-61.448,174.776,19.634,153.183
C03269=1086.004,61.059,-61.432,174.774,19.633,153.183
C03270=1085.998,60.810,-61.416,174.772,19.631,153.183
C03271=1085.993,60.560,-61.399,174.771,19.629,153.183
C03272=1085.987,60.311,-61.382,174.769,19.627,153.183
C03273=1085.981,60.062,-61.366,174.767,19.625,153.183
C03274=1085.975,59.812,-61.350,174.766,19.623,153.183
C03275=1085.969,59.563,-61.334,174.764,19.621,153.183
C03276=1085.964,59.313,-61.317,174.762,19.620,153.183
C03277=1085.958,59.064,-61.301,174.760,19.617,153.183
C03278=1085.952,58.815,-61.284,174.759,19.616,153.183
C03279=1085.946,58.565,-61.268,174.757,19.614,153.182
C03280=1085.940,58.316,-61.252,174.755,19.612,153.182
C03281=1085.935,58.066,-61.235,174.754,19.610,153.182
C03282=1085.929,57.817,-61.219,174.751,19.608,153.182
C03283=1085.923,57.568,-61.202,174.750,19.606,153.182
C03284=1085.917,57.318,-61.186,174.748,19.604,153.182
C03285=1085.911,57.068,-61.171,174.746,19.602,153.182
C03286=1085.905,56.819,-61.154,174.745,19.601,153.182
C03287=1085.900,56.569,-61.137,174.743,19.598,153.182
C03288=1085.894,56.320,-61.121,174.741,19.597,153.182
C03289=1085.889,56.071,-61.105,174.739,19.595,153.182
C03290=1085.883,55.822,-61.089,174.738,19.593,153.182
C03291=1085.877,55.573,-61.073,174.736,19.591,153.182
C03292=1085.871,55.323,-61.057,174.734,19.589,153.181
C03293=1085.865,55.073,-61.041,174.733,19.587,153.181
C03294=1085.860,54.824,-61.024,174.731,19.585,153.181
C03295=1085.854,54.574,-61.008,174.729,19.583,153.181
C03296=1085.848,54.325,-60.992,174.727,19.581,153.181
C03297=1085.842,54.076,-60.975,174.726,19.579,153.181
C03298=1085.837,53.827,-60.960,174.723,19.577,153.181
C03299=1085.831,53.577,-60.944,174.722,19.575,153.181
C03300=1085.825,53.328,-60.928,174.721,19.573,153.181
C03301=1085.819,53.078,-60.911,174.719,19.571,153.181
C03302=1085.814,52.829,-60.895,174.717,19.569,153.181
C03303=1085.808,52.579,-60.879,174.715,19.567,153.180
C03304=1085.803,52.330,-60.863,174.714,19.565,153.180
C03305=1085.797,52.081,-60.847,174.712,19.564,153.180
C03306=1085.791,51.831,-60.831,174.710,19.561,153.180
C03307=1085.785,51.581,-60.815,174.709,19.560,153.180
C03308=1085.779,51.332,-60.799,174.707,19.557,153.180
C03309=1085.774,51.083,-60.783,174.705,19.556,153.180
C03310=1085.768,50.834,-60.767,174.703,19.553,153.180
C03311=1085.763,50.584,-60.751,174.702,19.552,153.180
C03312=1085.757,50.335,-60.735,174.700,19.550,153.180
C03313=1085.751,50.085,-60.719,174.698,19.548,153.180
C03314=1085.746,49.835,-60.703,174.697,19.546,153.179
C03315=1085.740,49.586,-60.687,174.694,19.544,153.179
C03316=1085.734,49.337,-60.670,174.693,19.542,153.179
C03317=1085.729,49.087,-60.655,174.692,19.540,153.179
C03318=1085.723,48.838,-60.639,174.690,19.538,153.179
C03319=1085.717,48.589,-60.623,174.689,19.536,153.179
C03320=1085.712,48.339,-60.607,174.686,19.534,153.179
C03321=1085.706,48.090,-60.591,174.685,19.532,153.179
C03322=1085.700,47.840,-60.575,174.684,19.530,153.179
C03323=1085.694,47.562,-60.558,174.681,19.528,153.178
C03324=1085.688,47.283,-60.539,174.679,19.525,153.178
C03325=1085.681,47.005,-60.522,174.677,19.523,153.178
C03326=1085.675,46.727,-60.505,174.676,19.521,153.178
C03327=1085.669,46.478,-60.488,174.674,19.519,153.178
C03328=1085.664,46.228,-60.473,174.672,19.517,153.178
C03329=1085.658,45.978,-60.457,174.671,19.515,153.178
C03330=1085.653,45.729,-60.441,174.669,19.513,153.178
C03331=1085.647,45.480,-60.425,174.668,19.511,153.178
C03332=1085.641,45.230,-60.410,174.665,19.509,153.177
C03333=1085.636,44.981,-60.394,174.664,19.507,153.177
C03334=1085.630,44.731,-60.378,174.663,19.505,153.177
C03335=1085.624,44.482,-60.362,174.660,19.503,153.177
C03336=1085.619,44.232,-60.347,174.659,19.501,153.177
C03337=1085.613,43.983,-60.330,174.657,19.499,153.177
C03338=1085.607,43.733,-60.315,174.656,19.497,153.177
C03339=1085.602,43.484,-60.299,174.654,19.495,153.177
C03340=1085.596,43.234,-60.283,174.652,19.493,153.177
C03341=1085.591,42.985,-60.267,174.651,19.491,153.176
C03342=1085.584,42.735,-60.252,174.649,19.490,153.176
C03343=1085.579,42.487,-60.236,174.647,19.487,153.176
C03344=1085.573,42.237,-60.221,174.646,19.485,153.176
C03345=1085.568,41.987,-60.205,174.644,19.483,153.176
C03346=1085.562,41.738,-60.189,174.642,19.481,153.176
C03347=1085.556,41.489,-60.174,174.641,19.479,153.176
C03348=1085.550,41.239,-60.158,174.639,19.477,153.176
C03349=1085.544,40.989,-60.143,174.638,19.475,153.176
C03350=1085.539,40.740,-60.128,174.636,19.473,153.176
C03351=1085.533,40.491,-60.111,174.634,19.471,153.176
C03352=1085.527,40.241,-60.096,174.633,19.469,153.175
C03353=1085.521,39.992,-60.080,174.631,19.467,153.175
C03354=1085.516,39.742,-60.065,174.629,19.465,153.175
C03355=1085.510,39.492,-60.049,174.628,19.464,153.175
C03356=1085.505,39.244,-60.033,174.626,19.461,153.175
C03357=1085.498,38.994,-60.018,174.625,19.459,153.175
C03358=1085.493,38.744,-60.003,174.622,19.457,153.175
C03359=1085.488,38.495,-59.988,174.621,19.455,153.175
C03360=1085.482,38.246,-59.972,174.620,19.454,153.175
C03361=1085.476,37.997,-59.957,174.618,19.451,153.174
C03362=1085.470,37.747,-59.941,174.616,19.449,153.174
C03363=1085.464,37.497,-59.925,174.615,19.448,153.174
C03364=1085.458,37.248,-59.910,174.613,19.445,153.174
C03365=1085.453,36.998,-59.895,174.611,19.444,153.174
C03366=1085.447,36.748,-59.879,174.609,19.441,153.174
C03367=1085.441,36.499,-59.864,174.608,19.440,153.174
C03368=1085.436,36.250,-59.849,174.607,19.438,153.174
C03369=1085.429,36.000,-59.834,174.604,19.436,153.174
C03370=1085.424,35.751,-59.819,174.603,19.434,153.173
C03371=1085.418,35.502,-59.802,174.602,19.432,153.173
C03372=1085.412,35.252,-59.787,174.600,19.430,153.173
C03373=1085.407,35.003,-59.772,174.598,19.428,153.173
C03374=1085.400,34.753,-59.757,174.597,19.426,153.173
C03375=1085.395,34.503,-59.742,174.595,19.424,153.173
C03376=1085.389,34.255,-59.726,174.593,19.422,153.173
C03377=1085.383,34.005,-59.711,174.591,19.419,153.173
C03378=1085.378,33.756,-59.696,174.590,19.418,153.173
C03379=1085.372,33.506,-59.681,174.589,19.416,153.172
C03380=1085.366,33.256,-59.665,174.586,19.414,153.172
C03381=1085.360,33.007,-59.651,174.585,19.412,153.172
C03382=1085.355,32.757,-59.635,174.584,19.410,153.172
C03383=1085.349,32.508,-59.619,174.581,19.408,153.172
C03384=1085.343,32.259,-59.604,174.580,19.406,153.172
C03385=1085.337,32.009,-59.589,174.579,19.404,153.172
C03386=1085.331,31.760,-59.574,174.577,19.402,153.172
C03387=1085.325,31.481,-59.558,174.576,19.400,153.172
C03388=1085.319,31.203,-59.540,174.573,19.397,153.171
C03389=1085.312,30.924,-59.523,174.571,19.395,153.171
C03390=1085.306,30.646,-59.507,174.570,19.393,153.171
C03391=1085.300,30.397,-59.491,174.568,19.391,153.171
C03392=1085.294,30.147,-59.476,174.566,19.389,153.171
C03393=1085.289,29.898,-59.461,174.565,19.387,153.171
C03394=1085.283,29.649,-59.446,174.563,19.385,153.171
C03395=1085.277,29.399,-59.430,174.562,19.383,153.171
C03396=1085.271,29.150,-59.416,174.560,19.381,153.170
C03397=1085.266,28.900,-59.400,174.558,19.379,153.170
C03398=1085.260,28.651,-59.385,174.557,19.377,153.170
C03399=1085.254,28.401,-59.370,174.556,19.375,153.170
C03400=1085.248,28.152,-59.355,174.553,19.373,153.170
C03401=1085.242,27.902,-59.340,174.552,19.371,153.170
C03402=1085.237,27.653,-59.325,174.551,19.369,153.170
C03403=1085.231,27.403,-59.311,174.549,19.367,153.170
C03404=1085.226,27.153,-59.296,174.547,19.365,153.170
C03405=1085.219,26.904,-59.281,174.546,19.363,153.170
C03406=1085.214,26.655,-59.266,174.544,19.361,153.169
C03407=1085.208,26.405,-59.251,174.542,19.359,153.169
C03408=1085.202,26.156,-59.236,174.541,19.357,153.169
C03409=1085.197,25.906,-59.221,174.539,19.355,153.169
C03410=1085.190,25.656,-59.206,174.538,19.353,153.169
C03411=1085.184,25.407,-59.191,174.537,19.351,153.169
C03412=1085.179,25.157,-59.176,174.534,19.349,153.169
C03413=1085.173,24.908,-59.161,174.533,19.347,153.169
C03414=1085.167,24.659,-59.146,174.532,19.345,153.168
C03415=1085.162,24.409,-59.132,174.529,19.343,153.168
C03416=1085.156,24.159,-59.117,174.528,19.341,153.168
C03417=1085.150,23.910,-59.102,174.527,19.340,153.168
C03418=1085.144,23.660,-59.087,174.525,19.337,153.168
C03419=1085.138,23.411,-59.072,174.524,19.335,153.168
C03420=1085.133,23.162,-59.057,174.522,19.334,153.168
C03421=1085.127,22.912,-59.043,174.520,19.331,153.168
C03422=1085.121,22.663,-59.028,174.519,19.329,153.168
C03423=1085.115,22.413,-59.013,174.517,19.328,153.167
C03424=1085.109,22.164,-58.998,174.515,19.325,153.167
C03425=1085.104,21.914,-58.983,174.514,19.324,153.167
C03426=1085.098,21.665,-58.969,174.513,19.322,153.167
C03427=1085.092,21.415,-58.954,174.511,19.319,153.167
C03428=1085.087,21.166,-58.939,174.509,19.317,153.167
C03429=1085.080,20.916,-58.924,174.508,19.315,153.167
C03430=1085.075,20.666,-58.910,174.507,19.313,153.167
C03431=1085.069,20.417,-58.896,174.504,19.311,153.167
C03432=1085.063,20.167,-58.880,174.503,19.309,153.166
C03433=1085.058,19.919,-58.865,174.502,19.307,153.166
C03434=1085.052,19.668,-58.851,174.500,19.305,153.166
C03435=1085.046,19.419,-58.837,174.498,19.303,153.166
C03436=1085.040,19.169,-58.821,174.497,19.302,153.166
C03437=1085.035,18.920,-58.807,174.495,19.299,153.166
C03438=1085.029,18.671,-58.793,174.494,19.297,153.166
C03439=1085.022,18.421,-58.778,174.492,19.296,153.166
C03440=1085.017,18.172,-58.764,174.490,19.293,153.165
C03441=1085.011,17.922,-58.749,174.489,19.292,153.165
C03442=1085.006,17.673,-58.734,174.487,19.290,153.165
C03443=1085.000,17.423,-58.720,174.485,19.287,153.165
C03444=1084.994,17.173,-58.705,174.484,19.286,153.165
C03445=1084.988,16.924,-58.690,174.483,19.284,153.165
C03446=1084.982,16.674,-58.676,174.482,19.282,153.165
C03447=1084.976,16.425,-58.661,174.479,19.280,153.165
C03448=1084.971,16.175,-58.647,174.478,19.277,153.165
C03449=1084.965,15.926,-58.632,174.477,19.276,153.164
C03450=1084.959,15.677,-58.617,174.475,19.273,153.164
C03451=1084.953,15.399,-58.602,174.473,19.271,153.164
C03452=1084.946,15.123,-58.586,174.471,19.269,153.164
C03453=1084.940,14.845,-58.569,174.470,19.267,153.164
C03454=1084.933,14.568,-58.554,174.468,19.265,153.164
C03455=1084.928,14.319,-58.539,174.467,19.263,153.164
C03456=1084.922,14.070,-58.524,174.465,19.261,153.163
C03457=1084.916,13.820,-58.510,174.463,19.259,153.163
C03458=1084.910,13.571,-58.496,174.462,19.257,153.163
C03459=1084.904,13.321,-58.481,174.460,19.255,153.163
C03460=1084.898,13.072,-58.467,174.458,19.253,153.163
C03461=1084.893,12.822,-58.453,174.457,19.251,153.163
C03462=1084.886,12.572,-58.438,174.456,19.249,153.163
C03463=1084.881,12.323,-58.424,174.454,19.247,153.163
C03464=1084.875,12.074,-58.410,174.452,19.245,153.163
C03465=1084.869,11.824,-58.395,174.451,19.243,153.163
C03466=1084.863,11.575,-58.381,174.449,19.242,153.162
C03467=1084.857,11.324,-58.366,174.447,19.239,153.162
C03468=1084.851,11.076,-58.352,174.446,19.237,153.162
C03469=1084.845,10.826,-58.339,174.445,19.235,153.162
C03470=1084.839,10.576,-58.324,174.443,19.233,153.162
C03471=1084.833,10.327,-58.310,174.441,19.231,153.162
C03472=1084.828,10.077,-58.296,174.440,19.229,153.162
C03473=1084.821,9.828,-58.281,174.439,19.227,153.162
C03474=1084.816,9.578,-58.267,174.436,19.225,153.162
C03475=1084.810,9.329,-58.253,174.435,19.223,153.161
C03476=1084.804,9.079,-58.238,174.434,19.222,153.161
C03477=1084.798,8.829,-58.224,174.432,19.219,153.161
C03478=1084.793,8.580,-58.210,174.431,19.217,153.161
C03479=1084.787,8.330,-58.196,174.429,19.216,153.161
C03480=1084.780,8.081,-58.182,174.428,19.214,153.161
C03481=1084.775,7.832,-58.168,174.426,19.212,153.161
C03482=1084.769,7.582,-58.154,174.424,19.210,153.161
C03483=1084.763,7.332,-58.140,174.423,19.208,153.160
C03484=1084.757,7.083,-58.125,174.422,19.206,153.160
C03485=1084.752,6.833,-58.111,174.420,19.204,153.160
C03486=1084.746,6.583,-58.097,174.418,19.202,153.160
C03487=1084.740,6.334,-58.082,174.417,19.200,153.160
C03488=1084.734,6.085,-58.069,174.415,19.197,153.160
C03489=1084.728,5.835,-58.055,174.413,19.196,153.160
C03490=1084.722,5.586,-58.040,174.412,19.194,153.160
C03491=1084.716,5.336,-58.027,174.411,19.192,153.160
C03492=1084.711,5.087,-58.013,174.409,19.190,153.160
C03493=1084.705,4.837,-57.999,174.408,19.188,153.159
C03494=1084.699,4.587,-57.984,174.406,19.186,153.159
C03495=1084.694,4.338,-57.970,174.404,19.184,153.159
C03496=1084.687,4.089,-57.957,174.403,19.182,153.159
C03497=1084.682,3.839,-57.943,174.401,19.180,153.159
C03498=1084.676,3.589,-57.928,174.400,19.178,153.159
C03499=1084.670,3.340,-57.914,174.398,19.176,153.159
C03500=1084.665,3.090,-57.900,174.397,19.174,153.159
C03501=1084.659,2.841,-57.886,174.395,19.172,153.158
C03502=1084.653,2.591,-57.873,174.394,19.170,153.158
C03503=1084.647,2.342,-57.858,174.392,19.168,153.158
C03504=1084.641,2.092,-57.844,174.391,19.166,153.158
C03505=1084.636,1.843,-57.830,174.389,19.164,153.158
C03506=1084.630,1.593,-57.816,174.388,19.162,153.158
C03507=1084.625,1.343,-57.803,174.386,19.160,153.158
C03508=1084.618,1.093,-57.789,174.385,19.158,153.158
C03509=1084.612,0.844,-57.775,174.383,19.156,153.157
C03510=1084.607,0.595,-57.761,174.381,19.154,153.157
C03511=1084.601,0.345,-57.747,174.380,19.152,153.157
C03512=1084.596,0.096,-57.733,174.379,19.150,153.157
C03513=1084.589,-0.154,-57.720,174.378,19.148,153.157
C03514=1084.584,-0.403,-57.706,174.375,19.146,153.157
C03515=1084.577,-0.679,-57.690,174.374,19.144,153.157
C03516=1084.571,-0.954,-57.674,174.372,19.142,153.157
C03517=1084.565,-1.229,-57.659,174.371,19.140,153.156
C03518=1084.558,-1.504,-57.645,174.369,19.137,153.156
C03519=1084.553,-1.753,-57.631,174.367,19.135,153.156
C03520=1084.547,-2.003,-57.617,174.366,19.133,153.156
C03521=1084.541,-2.252,-57.604,174.365,19.131,153.156
C03522=1084.536,-2.502,-57.590,174.363,19.129,153.156
C03523=1084.530,-2.751,-57.575,174.361,19.127,153.156
C03524=1084.524,-3.000,-57.561,174.360,19.125,153.156
C03525=1084.518,-3.250,-57.548,174.359,19.124,153.155
C03526=1084.512,-3.500,-57.534,174.357,19.121,153.155
C03527=1084.506,-3.749,-57.520,174.355,19.120,153.155
C03528=1084.501,-3.999,-57.507,174.354,19.118,153.155
C03529=1084.495,-4.248,-57.493,174.353,19.116,153.155
C03530=1084.489,-4.497,-57.479,174.350,19.114,153.155
C03531=1084.483,-4.748,-57.465,174.349,19.112,153.155
C03532=1084.477,-4.998,-57.453,174.348,19.110,153.155
C03533=1084.471,-5.247,-57.439,174.347,19.108,153.155
C03534=1084.465,-5.496,-57.426,174.345,19.107,153.155
C03535=1084.460,-5.746,-57.412,174.343,19.104,153.154
C03536=1084.453,-5.995,-57.398,174.342,19.102,153.154
C03537=1084.448,-6.245,-57.385,174.340,19.100,153.154
C03538=1084.441,-6.495,-57.371,174.339,19.098,153.154
C03539=1084.436,-6.744,-57.357,174.337,19.096,153.154
C03540=1084.429,-6.994,-57.344,174.336,19.094,153.154
C03541=1084.424,-7.243,-57.330,174.334,19.093,153.154
C03542=1084.418,-7.492,-57.317,174.333,19.091,153.154
C03543=1084.412,-7.742,-57.303,174.331,19.089,153.154
C03544=1084.407,-7.992,-57.289,174.330,19.087,153.153
C03545=1084.401,-8.241,-57.276,174.328,19.085,153.153
C03546=1084.395,-8.491,-57.263,174.327,19.083,153.153
C03547=1084.389,-8.741,-57.249,174.325,19.081,153.153
C03548=1084.383,-8.991,-57.235,174.323,19.079,153.153
C03549=1084.377,-9.240,-57.222,174.322,19.077,153.153
C03550=1084.371,-9.489,-57.208,174.321,19.076,153.153
C03551=1084.366,-9.739,-57.195,174.320,19.073,153.153
C03552=1084.359,-9.989,-57.182,174.318,19.071,153.152
C03553=1084.354,-10.238,-57.168,174.316,19.069,153.152
C03554=1084.348,-10.487,-57.155,174.315,19.067,153.152
C03555=1084.342,-10.737,-57.141,174.313,19.066,153.152
C03556=1084.336,-10.987,-57.129,174.311,19.063,153.152
C03557=1084.331,-11.236,-57.115,174.310,19.062,153.152
C03558=1084.325,-11.486,-57.101,174.309,19.060,153.152
C03559=1084.319,-11.735,-57.088,174.308,19.058,153.152
C03560=1084.313,-11.985,-57.074,174.305,19.056,153.152
C03561=1084.308,-12.235,-57.061,174.304,19.054,153.151
C03562=1084.302,-12.484,-57.048,174.303,19.052,153.151
C03563=1084.296,-12.734,-57.034,174.301,19.050,153.151
C03564=1084.290,-12.983,-57.021,174.300,19.048,153.151
C03565=1084.284,-13.233,-57.008,174.298,19.046,153.151
C03566=1084.278,-13.482,-56.994,174.297,19.044,153.151
C03567=1084.272,-13.732,-56.981,174.295,19.042,153.151
C03568=1084.267,-13.982,-56.968,174.294,19.040,153.151
C03569=1084.261,-14.231,-56.955,174.292,19.038,153.151
C03570=1084.255,-14.481,-56.941,174.291,19.036,153.151
C03571=1084.249,-14.730,-56.928,174.289,19.034,153.150
C03572=1084.243,-14.980,-56.915,174.288,19.033,153.150
C03573=1084.238,-15.229,-56.901,174.287,19.031,153.150
C03574=1084.232,-15.479,-56.888,174.284,19.029,153.150
C03575=1084.226,-15.728,-56.875,174.283,19.027,153.150
C03576=1084.220,-15.978,-56.861,174.282,19.025,153.150
C03577=1084.214,-16.228,-56.849,174.281,19.023,153.150
C03578=1084.208,-16.477,-56.836,174.279,19.022,153.150
C03579=1084.201,-16.751,-56.821,174.277,19.019,153.150
C03580=1084.195,-17.025,-56.807,174.276,19.017,153.150
C03581=1084.188,-17.298,-56.792,174.274,19.015,153.149
C03582=1084.182,-17.571,-56.778,174.272,19.013,153.149
C03583=1084.176,-17.820,-56.764,174.271,19.011,153.149
C03584=1084.170,-18.070,-56.752,174.269,19.009,153.149
C03585=1084.164,-18.319,-56.738,174.268,19.007,153.149
C03586=1084.158,-18.569,-56.726,174.266,19.005,153.149
C03587=1084.152,-18.819,-56.713,174.265,19.004,153.149
C03588=1084.147,-19.069,-56.699,174.264,19.002,153.149
C03589=1084.141,-19.318,-56.686,174.261,19.000,153.149
C03590=1084.135,-19.567,-56.673,174.260,18.998,153.148
C03591=1084.129,-19.817,-56.660,174.259,18.996,153.148
C03592=1084.123,-20.067,-56.647,174.258,18.994,153.148
C03593=1084.117,-20.317,-56.634,174.256,18.993,153.148
C03594=1084.111,-20.566,-56.621,174.254,18.990,153.148
C03595=1084.105,-20.816,-56.608,174.253,18.988,153.148
C03596=1084.099,-21.065,-56.595,174.251,18.986,153.148
C03597=1084.094,-21.315,-56.582,174.250,18.985,153.148
C03598=1084.087,-21.564,-56.568,174.249,18.983,153.148
C03599=1084.082,-21.814,-56.556,174.246,18.981,153.148
C03600=1084.076,-22.063,-56.543,174.245,18.979,153.147
C03601=1084.070,-22.313,-56.530,174.244,18.977,153.147
C03602=1084.065,-22.563,-56.517,174.243,18.975,153.147
C03603=1084.059,-22.812,-56.504,174.241,18.974,153.147
C03604=1084.053,-23.062,-56.491,174.239,18.971,153.147
C03605=1084.047,-23.311,-56.478,174.238,18.970,153.147
C03606=1084.041,-23.561,-56.466,174.237,18.968,153.147
C03607=1084.034,-23.811,-56.452,174.235,18.966,153.147
C03608=1084.029,-24.061,-56.439,174.234,18.964,153.147
C03609=1084.024,-24.310,-56.427,174.232,18.962,153.147
C03610=1084.018,-24.559,-56.414,174.230,18.960,153.146
C03611=1084.012,-24.809,-56.401,174.229,18.958,153.146
C03612=1084.006,-25.059,-56.389,174.228,18.956,153.146
C03613=1084.000,-25.308,-56.375,174.226,18.955,153.146
C03614=1083.994,-25.558,-56.363,174.225,18.953,153.146
C03615=1083.988,-25.808,-56.349,174.223,18.951,153.146
C03616=1083.982,-26.058,-56.336,174.222,18.949,153.146
C03617=1083.977,-26.307,-56.324,174.220,18.947,153.146
C03618=1083.971,-26.556,-56.311,174.219,18.945,153.146
C03619=1083.965,-26.806,-56.298,174.218,18.944,153.146
C03620=1083.959,-27.056,-56.286,174.216,18.942,153.145
C03621=1083.953,-27.305,-56.273,174.214,18.939,153.145
C03622=1083.947,-27.555,-56.260,174.213,18.938,153.145
C03623=1083.941,-27.805,-56.247,174.211,18.936,153.145
C03624=1083.936,-28.054,-56.235,174.210,18.934,153.145
C03625=1083.930,-28.303,-56.222,174.209,18.932,153.145
C03626=1083.924,-28.553,-56.209,174.207,18.930,153.145
C03627=1083.918,-28.803,-56.197,174.205,18.929,153.145
C03628=1083.912,-29.052,-56.184,174.204,18.927,153.145
C03629=1083.906,-29.302,-56.171,174.202,18.925,153.145
C03630=1083.900,-29.552,-56.159,174.201,18.923,153.145
C03631=1083.894,-29.802,-56.146,174.200,18.922,153.145
C03632=1083.888,-30.050,-56.133,174.198,18.920,153.145
C03633=1083.882,-30.300,-56.121,174.196,18.918,153.144
C03634=1083.876,-30.550,-56.108,174.195,18.916,153.144
C03635=1083.870,-30.800,-56.096,174.194,18.914,153.144
C03636=1083.864,-31.050,-56.083,174.192,18.912,153.144
C03637=1083.858,-31.299,-56.070,174.191,18.911,153.144
